LIN {X 0,Y 523.95,Z 619.34,A -85,B 0,C 180,E1 -4877.97,E2 -4877.97} C_VEL
LIN {X 0,Y 523.975,Z 619.339,A -85,B 0,C 180,E1 -4880.41,E2 -4880.41} C_VEL
LIN {X 0,Y 523.913,Z 619.349,A -85,B 0,C 180,E1 -4882.894,E2 -4882.894} C_VEL
LIN {X 0,Y 523.937,Z 619.342,A -85,B 0,C 180,E1 -4885.42,E2 -4885.42} C_VEL
LIN {X 0,Y 523.92,Z 619.339,A -85,B 0,C 180,E1 -4888.002,E2 -4888.002} C_VEL
LIN {X 0,Y 523.942,Z 619.344,A -85,B 0,C 180,E1 -4890.854,E2 -4890.854} C_VEL
LIN {X 0,Y 523.932,Z 619.34,A -85,B 0,C 180,E1 -4893.73,E2 -4893.73} C_VEL
LIN {X 0,Y 523.906,Z 619.346,A -85,B 0,C 180,E1 -4896.401,E2 -4896.401} C_VEL
LIN {X 0,Y 523.915,Z 619.351,A -85,B 0,C 180,E1 -4899.086,E2 -4899.086} C_VEL
LIN {X 0,Y 523.91,Z 619.344,A -85,B 0,C 180,E1 -4902.124,E2 -4902.124} C_VEL
LIN {X 0,Y 523.939,Z 619.346,A -85,B 0,C 180,E1 -4905.311,E2 -4905.311} C_VEL
LIN {X 0,Y 523.883,Z 619.351,A -85,B 0,C 180,E1 -4906.91,E2 -4906.91} C_VEL
LIN {X 0,Y 523.204,Z 619.439,A -85,B 0,C 180,E1 -4907.552,E2 -4907.552} C_VEL
LIN {X 0,Y 520.358,Z 619.789,A -85,B 0,C 180,E1 -4908.594,E2 -4908.594} C_VEL
LIN {X 0,Y 517.964,Z 620.093,A -85,B 0,C 180,E1 -4909.433,E2 -4909.433} C_VEL
LIN {X 0,Y 516.942,Z 620.215,A -85,B 0,C 180,E1 -4910.08,E2 -4910.08} C_VEL
LIN {X 0,Y 516.861,Z 620.224,A -85,B 0,C 180,E1 -4910.3,E2 -4910.3} C_VEL
LIN {X 0,Y 516.879,Z 620.229,A -85,B 0,C 180,E1 -4913.344,E2 -4913.344} C_VEL
LIN {X 0,Y 516.883,Z 620.22,A -85,B 0,C 180,E1 -4916.119,E2 -4916.119} C_VEL
LIN {X 0,Y 516.884,Z 620.224,A -85,B 0,C 180,E1 -4918.938,E2 -4918.938} C_VEL
LIN {X 0,Y 516.851,Z 620.232,A -85,B 0,C 180,E1 -4921.581,E2 -4921.581} C_VEL
LIN {X 0,Y 516.897,Z 620.309,A -85,B 0,C 180,E1 -4922.931,E2 -4922.931} C_VEL
LIN {X 0,Y 518.133,Z 627.417,A -85,B 0,C 180,E1 -4924.275,E2 -4924.275} C_VEL
LIN {X 0,Y 517.808,Z 639.497,A -85,B 0,C 180,E1 -4926.421,E2 -4926.421} C_VEL
LIN {X 0,Y 520.426,Z 652.346,A -85,B 0,C 180,E1 -4926.713,E2 -4926.713} C_VEL
LIN {X 0,Y 519.719,Z 775.501,A -85,B 0,C 180,E1 -4928.455,E2 -4928.455} C_VEL
LIN {X 0,Y 519.426,Z 789.891,A -85,B 0,C 180,E1 -4928.813,E2 -4928.813} C_VEL
LIN {X 0,Y 519.114,Z 803.721,A -85,B 0,C 180,E1 -4929.322,E2 -4929.322} C_VEL
LIN {X 0,Y 518.734,Z 817.355,A -85,B 0,C 180,E1 -4929.995,E2 -4929.995} C_VEL
LIN {X 0,Y 518.294,Z 830.118,A -85,B 0,C 180,E1 -4930.802,E2 -4930.802} C_VEL
LIN {X 0,Y 517.887,Z 841.924,A -85,B 0,C 180,E1 -4931.73,E2 -4931.73} C_VEL
LIN {X 0,Y 517.463,Z 853.262,A -85,B 0,C 180,E1 -4932.818,E2 -4932.818} C_VEL
LIN {X 0,Y 517.098,Z 863.506,A -85,B 0,C 180,E1 -4934.025,E2 -4934.025} C_VEL
LIN {X 0,Y 516.77,Z 873.237,A -85,B 0,C 180,E1 -4935.428,E2 -4935.428} C_VEL
LIN {X 0,Y 516.533,Z 881.108,A -85,B 0,C 180,E1 -4936.826,E2 -4936.826} C_VEL
LIN {X 0,Y 516.373,Z 887.392,A -85,B 0,C 180,E1 -4938.22,E2 -4938.22} C_VEL
LIN {X 0,Y 516.321,Z 891.674,A -85,B 0,C 180,E1 -4939.411,E2 -4939.411} C_VEL
LIN {X 0,Y 516.246,Z 895.077,A -85,B 0,C 180,E1 -4940.598,E2 -4940.598} C_VEL
LIN {X 0,Y 516.232,Z 898.246,A -85,B 0,C 180,E1 -4942.176,E2 -4942.176} C_VEL
LIN {X 0,Y 516.254,Z 900.019,A -85,B 0,C 180,E1 -4943.748,E2 -4943.748} C_VEL
LIN {X 0,Y 516.211,Z 900.451,A -85,B 0,C 180,E1 -4945.314,E2 -4945.314} C_VEL
LIN {X 0,Y 516.265,Z 899.556,A -85,B 0,C 180,E1 -4946.879,E2 -4946.879} C_VEL
LIN {X 0,Y 516.195,Z 897.325,A -85,B 0,C 180,E1 -4948.44,E2 -4948.44} C_VEL
LIN {X 0,Y 516.205,Z 893.711,A -85,B 0,C 180,E1 -4950,E2 -4950} C_VEL
LIN {X 0,Y 516.38,Z 890.026,A -85,B 0,C 180,E1 -4951.17,E2 -4951.17} C_VEL
LIN {X 0,Y 516.369,Z 885.463,A -85,B 0,C 180,E1 -4952.34,E2 -4952.34} C_VEL
LIN {X 0,Y 516.636,Z 878.835,A -85,B 0,C 180,E1 -4953.705,E2 -4953.705} C_VEL
LIN {X 0,Y 516.886,Z 870.62,A -85,B 0,C 180,E1 -4955.07,E2 -4955.07} C_VEL
LIN {X 0,Y 517.131,Z 862.132,A -85,B 0,C 180,E1 -4956.242,E2 -4956.242} C_VEL
LIN {X 0,Y 517.523,Z 851.815,A -85,B 0,C 180,E1 -4957.419,E2 -4957.419} C_VEL
LIN {X 0,Y 517.941,Z 840.432,A -85,B 0,C 180,E1 -4958.486,E2 -4958.486} C_VEL
LIN {X 0,Y 518.356,Z 829.005,A -85,B 0,C 180,E1 -4959.364,E2 -4959.364} C_VEL
LIN {X 0,Y 518.753,Z 816.473,A -85,B 0,C 180,E1 -4960.144,E2 -4960.144} C_VEL
LIN {X 0,Y 519.16,Z 803.502,A -85,B 0,C 180,E1 -4960.777,E2 -4960.777} C_VEL
LIN {X 0,Y 519.429,Z 789.513,A -85,B 0,C 180,E1 -4961.29,E2 -4961.29} C_VEL
LIN {X 0,Y 519.647,Z 775.805,A -85,B 0,C 180,E1 -4961.631,E2 -4961.631} C_VEL
LIN {X 0,Y 520.391,Z 652.06,A -85,B 0,C 180,E1 -4963.382,E2 -4963.382} C_VEL
LIN {X 0,Y 517.871,Z 639.491,A -85,B 0,C 180,E1 -4963.663,E2 -4963.663} C_VEL
LIN {X 0,Y 518.127,Z 626.693,A -85,B 0,C 180,E1 -4965.943,E2 -4965.943} C_VEL
LIN {X 0,Y 516.901,Z 620.224,A -85,B 0,C 180,E1 -4967.201,E2 -4967.201} C_VEL
LIN {X 0,Y 516.934,Z 620.221,A -85,B 0,C 180,E1 -4970.265,E2 -4970.265} C_VEL
LIN {X 0,Y 516.86,Z 620.226,A -85,B 0,C 180,E1 -4973.224,E2 -4973.224} C_VEL
LIN {X 0,Y 516.859,Z 620.226,A -85,B 0,C 180,E1 -4976.176,E2 -4976.176} C_VEL
LIN {X 0,Y 516.902,Z 620.22,A -85,B 0,C 180,E1 -4979.306,E2 -4979.306} C_VEL
LIN {X 0,Y 516.867,Z 620.227,A -85,B 0,C 180,E1 -4982.537,E2 -4982.537} C_VEL
LIN {X 0,Y 516.854,Z 620.226,A -85,B 0,C 180,E1 -4985.327,E2 -4985.327} C_VEL
LIN {X 0,Y 516.872,Z 620.227,A -85,B 0,C 180,E1 -4988.717,E2 -4988.717} C_VEL
LIN {X 0,Y 516.848,Z 620.224,A -85,B 0,C 180,E1 -4991.782,E2 -4991.782} C_VEL
LIN {X 0,Y 516.899,Z 620.225,A -85,B 0,C 180,E1 -4995.007,E2 -4995.007} C_VEL
LIN {X 0,Y 516.853,Z 620.224,A -85,B 0,C 180,E1 -4998.407,E2 -4998.407} C_VEL
LIN {X 0,Y 516.874,Z 620.221,A -85,B 0,C 180,E1 -5001.283,E2 -5001.283} C_VEL
LIN {X 0,Y 516.863,Z 620.22,A -85,B 0,C 180,E1 -5004.671,E2 -5004.671} C_VEL
LIN {X 0,Y 516.897,Z 620.223,A -85,B 0,C 180,E1 -5007.457,E2 -5007.457} C_VEL
LIN {X 0,Y 516.922,Z 620.213,A -85,B 0,C 180,E1 -5010.695,E2 -5010.695} C_VEL
LIN {X 0,Y 516.882,Z 620.221,A -85,B 0,C 180,E1 -5013.818,E2 -5013.818} C_VEL
LIN {X 0,Y 516.861,Z 620.22,A -85,B 0,C 180,E1 -5016.776,E2 -5016.776} C_VEL
LIN {X 0,Y 516.943,Z 620.216,A -85,B 0,C 180,E1 -5019.732,E2 -5019.732} C_VEL
LIN {X 0,Y 516.909,Z 620.21,A -85,B 0,C 180,E1 -5022.595,E2 -5022.595} C_VEL
LIN {X 0,Y 516.946,Z 620.213,A -85,B 0,C 180,E1 -5025.03,E2 -5025.03} C_VEL
LIN {X 0,Y 516.97,Z 620.207,A -85,B 0,C 180,E1 -5028.233,E2 -5028.233} C_VEL
LIN {X 0,Y 516.967,Z 620.211,A -85,B 0,C 180,E1 -5031.399,E2 -5031.399} C_VEL
LIN {X 0,Y 517.017,Z 620.202,A -85,B 0,C 180,E1 -5034.54,E2 -5034.54} C_VEL
LIN {X 0,Y 517.084,Z 620.201,A -85,B 0,C 180,E1 -5037.663,E2 -5037.663} C_VEL
LIN {X 0,Y 517.094,Z 620.19,A -85,B 0,C 180,E1 -5040.779,E2 -5040.779} C_VEL
LIN {X 0,Y 517.012,Z 620.204,A -85,B 0,C 180,E1 -5043.117,E2 -5043.117} C_VEL
LIN {X 0,Y 516.995,Z 620.209,A -85,B 0,C 180,E1 -5046.243,E2 -5046.243} C_VEL
LIN {X 0,Y 516.968,Z 620.21,A -85,B 0,C 180,E1 -5048.6,E2 -5048.6} C_VEL
LIN {X 0,Y 516.956,Z 620.215,A -85,B 0,C 180,E1 -5051.807,E2 -5051.807} C_VEL
LIN {X 0,Y 516.948,Z 620.209,A -85,B 0,C 180,E1 -5055.146,E2 -5055.146} C_VEL
LIN {X 0,Y 516.928,Z 620.22,A -85,B 0,C 180,E1 -5058.222,E2 -5058.222} C_VEL
LIN {X 0,Y 516.915,Z 620.216,A -85,B 0,C 180,E1 -5060.701,E2 -5060.701} C_VEL
LIN {X 0,Y 516.893,Z 620.224,A -85,B 0,C 180,E1 -5064.073,E2 -5064.073} C_VEL
LIN {X 0,Y 516.927,Z 620.215,A -85,B 0,C 180,E1 -5066.658,E2 -5066.658} C_VEL
LIN {X 0,Y 516.914,Z 620.216,A -85,B 0,C 180,E1 -5069.524,E2 -5069.524} C_VEL
LIN {X 0,Y 516.9,Z 620.223,A -85,B 0,C 180,E1 -5072.544,E2 -5072.544} C_VEL
LIN {X 0,Y 516.869,Z 620.221,A -85,B 0,C 180,E1 -5075.33,E2 -5075.33} C_VEL
LIN {X 0,Y 516.884,Z 620.222,A -85,B 0,C 180,E1 -5077.943,E2 -5077.943} C_VEL
LIN {X 0,Y 516.905,Z 620.222,A -85,B 0,C 180,E1 -5080.74,E2 -5080.74} C_VEL
LIN {X 0,Y 516.885,Z 620.22,A -85,B 0,C 180,E1 -5083.903,E2 -5083.903} C_VEL
LIN {X 0,Y 516.884,Z 620.222,A -85,B 0,C 180,E1 -5086.107,E2 -5086.107} C_VEL
LIN {X 0,Y 516.92,Z 620.221,A -85,B 0,C 180,E1 -5088.398,E2 -5088.398} C_VEL
LIN {X 0,Y 516.883,Z 620.222,A -85,B 0,C 180,E1 -5091.284,E2 -5091.284} C_VEL
LIN {X 0,Y 516.893,Z 620.222,A -85,B 0,C 180,E1 -5094.221,E2 -5094.221} C_VEL
LIN {X 0,Y 516.9,Z 620.223,A -85,B 0,C 180,E1 -5097.053,E2 -5097.053} C_VEL
LIN {X 0,Y 516.895,Z 620.221,A -85,B 0,C 180,E1 -5099.796,E2 -5099.796} C_VEL
LIN {X 0,Y 516.93,Z 620.22,A -85,B 0,C 180,E1 -5102.906,E2 -5102.906} C_VEL
LIN {X 0,Y 516.982,Z 620.308,A -85,B 0,C 180,E1 -5103.318,E2 -5103.318} C_VEL
LIN {X 0,Y 519.43,Z 632.291,A -85,B 0,C 180,E1 -5105.201,E2 -5105.201} C_VEL
LIN {X 0,Y 518.76,Z 652.815,A -85,B 0,C 180,E1 -5108.126,E2 -5108.126} C_VEL
LIN {X 0,Y 518.152,Z 675.928,A -85,B 0,C 180,E1 -5111.374,E2 -5111.374} C_VEL
LIN {X 0,Y 520.468,Z 690.281,A -85,B 0,C 180,E1 -5111.668,E2 -5111.668} C_VEL
LIN {X 0,Y 519.629,Z 814.592,A -85,B 0,C 180,E1 -5113.423,E2 -5113.423} C_VEL
LIN {X 0,Y 519.394,Z 829.055,A -85,B 0,C 180,E1 -5113.792,E2 -5113.792} C_VEL
LIN {X 0,Y 519.121,Z 842.489,A -85,B 0,C 180,E1 -5114.29,E2 -5114.29} C_VEL
LIN {X 0,Y 518.758,Z 854.701,A -85,B 0,C 180,E1 -5114.883,E2 -5114.883} C_VEL
LIN {X 0,Y 518.28,Z 867.555,A -85,B 0,C 180,E1 -5115.672,E2 -5115.672} C_VEL
LIN {X 0,Y 517.884,Z 879.251,A -85,B 0,C 180,E1 -5116.562,E2 -5116.562} C_VEL
LIN {X 0,Y 517.561,Z 888.983,A -85,B 0,C 180,E1 -5117.451,E2 -5117.451} C_VEL
LIN {X 0,Y 517.252,Z 899.705,A -85,B 0,C 180,E1 -5118.637,E2 -5118.637} C_VEL
LIN {X 0,Y 516.88,Z 908.555,A -85,B 0,C 180,E1 -5119.819,E2 -5119.819} C_VEL
LIN {X 0,Y 516.689,Z 915.917,A -85,B 0,C 180,E1 -5121.001,E2 -5121.001} C_VEL
LIN {X 0,Y 516.501,Z 922.054,A -85,B 0,C 180,E1 -5122.179,E2 -5122.179} C_VEL
LIN {X 0,Y 516.395,Z 928.568,A -85,B 0,C 180,E1 -5123.749,E2 -5123.749} C_VEL
LIN {X 0,Y 516.305,Z 932.38,A -85,B 0,C 180,E1 -5124.924,E2 -5124.924} C_VEL
LIN {X 0,Y 516.325,Z 935.316,A -85,B 0,C 180,E1 -5126.097,E2 -5126.097} C_VEL
LIN {X 0,Y 516.258,Z 938.002,A -85,B 0,C 180,E1 -5127.659,E2 -5127.659} C_VEL
LIN {X 0,Y 516.155,Z 939.334,A -85,B 0,C 180,E1 -5129.22,E2 -5129.22} C_VEL
LIN {X 0,Y 516.155,Z 939.334,A -85,B 0,C 180,E1 -5130.78,E2 -5130.78} C_VEL
LIN {X 0,Y 516.258,Z 938.005,A -85,B 0,C 180,E1 -5132.341,E2 -5132.341} C_VEL
LIN {X 0,Y 516.325,Z 935.32,A -85,B 0,C 180,E1 -5133.902,E2 -5133.902} C_VEL
LIN {X 0,Y 516.388,Z 931.201,A -85,B 0,C 180,E1 -5135.467,E2 -5135.467} C_VEL
LIN {X 0,Y 516.406,Z 925.526,A -85,B 0,C 180,E1 -5137.035,E2 -5137.035} C_VEL
LIN {X 0,Y 516.599,Z 919.127,A -85,B 0,C 180,E1 -5138.409,E2 -5138.409} C_VEL
LIN {X 0,Y 516.826,Z 911.174,A -85,B 0,C 180,E1 -5139.787,E2 -5139.787} C_VEL
LIN {X 0,Y 517.109,Z 902.852,A -85,B 0,C 180,E1 -5140.969,E2 -5140.969} C_VEL
LIN {X 0,Y 517.455,Z 892.433,A -85,B 0,C 180,E1 -5142.197,E2 -5142.197} C_VEL
LIN {X 0,Y 517.808,Z 881.609,A -85,B 0,C 180,E1 -5143.24,E2 -5143.24} C_VEL
LIN {X 0,Y 518.211,Z 870.422,A -85,B 0,C 180,E1 -5144.13,E2 -5144.13} C_VEL
LIN {X 0,Y 518.634,Z 858.246,A -85,B 0,C 180,E1 -5144.92,E2 -5144.92} C_VEL
LIN {X 0,Y 519.026,Z 844.741,A -85,B 0,C 180,E1 -5145.612,E2 -5145.612} C_VEL
LIN {X 0,Y 519.364,Z 830.319,A -85,B 0,C 180,E1 -5146.166,E2 -5146.166} C_VEL
LIN {X 0,Y 519.645,Z 815.731,A -85,B 0,C 180,E1 -5146.551,E2 -5146.551} C_VEL
LIN {X 0,Y 519.827,Z 787.602,A -85,B 0,C 180,E1 -5146.974,E2 -5146.974} C_VEL
LIN {X 0,Y 520.385,Z 688.558,A -85,B 0,C 180,E1 -5148.359,E2 -5148.359} C_VEL
LIN {X 0,Y 518.155,Z 675.916,A -85,B 0,C 180,E1 -5148.626,E2 -5148.626} C_VEL
LIN {X 0,Y 518.806,Z 651.311,A -85,B 0,C 180,E1 -5152.081,E2 -5152.081} C_VEL
LIN {X 0,Y 519.377,Z 633.721,A -85,B 0,C 180,E1 -5154.588,E2 -5154.588} C_VEL
LIN {X 0,Y 518.926,Z 629.314,A -85,B 0,C 180,E1 -5155.253,E2 -5155.253} C_VEL
LIN {X 0,Y 516.965,Z 620.217,A -85,B 0,C 180,E1 -5156.71,E2 -5156.71} C_VEL
LIN {X 0,Y 516.913,Z 620.223,A -85,B 0,C 180,E1 -5159.524,E2 -5159.524} C_VEL
LIN {X 0,Y 516.902,Z 620.218,A -85,B 0,C 180,E1 -5162.544,E2 -5162.544} C_VEL
LIN {X 0,Y 516.885,Z 620.224,A -85,B 0,C 180,E1 -5165.332,E2 -5165.332} C_VEL
LIN {X 0,Y 516.886,Z 620.221,A -85,B 0,C 180,E1 -5167.944,E2 -5167.944} C_VEL
LIN {X 0,Y 516.887,Z 620.218,A -85,B 0,C 180,E1 -5170.741,E2 -5170.741} C_VEL
LIN {X 0,Y 516.905,Z 620.219,A -85,B 0,C 180,E1 -5172.829,E2 -5172.829} C_VEL
LIN {X 0,Y 516.924,Z 620.215,A -85,B 0,C 180,E1 -5175.01,E2 -5175.01} C_VEL
LIN {X 0,Y 516.924,Z 620.212,A -85,B 0,C 180,E1 -5178.398,E2 -5178.398} C_VEL
LIN {X 0,Y 516.888,Z 620.224,A -85,B 0,C 180,E1 -5181.285,E2 -5181.285} C_VEL
LIN {X 0,Y 516.893,Z 620.22,A -85,B 0,C 180,E1 -5184.221,E2 -5184.221} C_VEL
LIN {X 0,Y 516.899,Z 620.217,A -85,B 0,C 180,E1 -5187.053,E2 -5187.053} C_VEL
LIN {X 0,Y 516.894,Z 620.22,A -85,B 0,C 180,E1 -5189.797,E2 -5189.797} C_VEL
LIN {X 0,Y 516.93,Z 620.214,A -85,B 0,C 180,E1 -5192.468,E2 -5192.468} C_VEL
LIN {X 0,Y 516.912,Z 620.215,A -85,B 0,C 180,E1 -5195.072,E2 -5195.072} C_VEL
LIN {X 0,Y 516.872,Z 620.224,A -85,B 0,C 180,E1 -5197.622,E2 -5197.622} C_VEL
LIN {X 0,Y 516.934,Z 620.219,A -85,B 0,C 180,E1 -5200.13,E2 -5200.13} C_VEL
LIN {X 0,Y 516.933,Z 620.214,A -85,B 0,C 180,E1 -5202.596,E2 -5202.596} C_VEL
LIN {X 0,Y 516.944,Z 620.211,A -85,B 0,C 180,E1 -5205.03,E2 -5205.03} C_VEL
LIN {X 0,Y 516.968,Z 620.217,A -85,B 0,C 180,E1 -5208.234,E2 -5208.234} C_VEL
LIN {X 0,Y 516.97,Z 620.206,A -85,B 0,C 180,E1 -5211.4,E2 -5211.4} C_VEL
LIN {X 0,Y 517.011,Z 620.207,A -85,B 0,C 180,E1 -5213.757,E2 -5213.757} C_VEL
LIN {X 0,Y 517.085,Z 620.195,A -85,B 0,C 180,E1 -5217.663,E2 -5217.663} C_VEL
LIN {X 0,Y 517.094,Z 620.195,A -85,B 0,C 180,E1 -5220.779,E2 -5220.779} C_VEL
LIN {X 0,Y 517.013,Z 620.204,A -85,B 0,C 180,E1 -5223.117,E2 -5223.117} C_VEL
LIN {X 0,Y 517.004,Z 620.207,A -85,B 0,C 180,E1 -5226.243,E2 -5226.243} C_VEL
LIN {X 0,Y 516.946,Z 620.21,A -85,B 0,C 180,E1 -5229.39,E2 -5229.39} C_VEL
LIN {X 0,Y 516.955,Z 620.21,A -85,B 0,C 180,E1 -5231.807,E2 -5231.807} C_VEL
LIN {X 0,Y 516.95,Z 620.212,A -85,B 0,C 180,E1 -5235.148,E2 -5235.148} C_VEL
LIN {X 0,Y 516.919,Z 620.218,A -85,B 0,C 180,E1 -5238.223,E2 -5238.223} C_VEL
LIN {X 0,Y 516.915,Z 620.223,A -85,B 0,C 180,E1 -5240.702,E2 -5240.702} C_VEL
LIN {X 0,Y 516.904,Z 620.216,A -85,B 0,C 180,E1 -5244.073,E2 -5244.073} C_VEL
LIN {X 0,Y 516.9,Z 620.224,A -85,B 0,C 180,E1 -5246.66,E2 -5246.66} C_VEL
LIN {X 0,Y 516.911,Z 620.212,A -85,B 0,C 180,E1 -5249.523,E2 -5249.523} C_VEL
LIN {X 0,Y 516.897,Z 620.222,A -85,B 0,C 180,E1 -5252.543,E2 -5252.543} C_VEL
LIN {X 0,Y 516.868,Z 620.226,A -85,B 0,C 180,E1 -5255.33,E2 -5255.33} C_VEL
LIN {X 0,Y 516.881,Z 620.22,A -85,B 0,C 180,E1 -5257.943,E2 -5257.943} C_VEL
LIN {X 0,Y 516.856,Z 620.225,A -85,B 0,C 180,E1 -5260.745,E2 -5260.745} C_VEL
LIN {X 0,Y 516.883,Z 620.221,A -85,B 0,C 180,E1 -5263.904,E2 -5263.904} C_VEL
LIN {X 0,Y 516.839,Z 620.23,A -85,B 0,C 180,E1 -5266.911,E2 -5266.911} C_VEL
LIN {X 0,Y 516.862,Z 620.229,A -85,B 0,C 180,E1 -5269.593,E2 -5269.593} C_VEL
LIN {X 0,Y 516.861,Z 620.224,A -85,B 0,C 180,E1 -5270.3,E2 -5270.3} C_VEL
LIN {X 0,Y 516.204,Z 620.312,A -85,B 0,C 180,E1 -5270.95,E2 -5270.95} C_VEL
LIN {X 0,Y 513.367,Z 620.666,A -85,B 0,C 180,E1 -5272.006,E2 -5272.006} C_VEL
LIN {X 0,Y 510.957,Z 620.967,A -85,B 0,C 180,E1 -5272.856,E2 -5272.856} C_VEL
LIN {X 0,Y 509.912,Z 621.094,A -85,B 0,C 180,E1 -5273.513,E2 -5273.513} C_VEL
LIN {X 0,Y 509.821,Z 621.102,A -85,B 0,C 180,E1 -5273.736,E2 -5273.736} C_VEL
LIN {X 0,Y 509.842,Z 621.097,A -85,B 0,C 180,E1 -5276.538,E2 -5276.538} C_VEL
LIN {X 0,Y 509.832,Z 621.106,A -85,B 0,C 180,E1 -5279.333,E2 -5279.333} C_VEL
LIN {X 0,Y 509.856,Z 621.101,A -85,B 0,C 180,E1 -5282.498,E2 -5282.498} C_VEL
LIN {X 0,Y 509.852,Z 621.138,A -85,B 0,C 180,E1 -5282.721,E2 -5282.721} C_VEL
LIN {X 0,Y 511.174,Z 628.426,A -85,B 0,C 180,E1 -5284.118,E2 -5284.118} C_VEL
LIN {X 0,Y 510.904,Z 639.791,A -85,B 0,C 180,E1 -5286.162,E2 -5286.162} C_VEL
LIN {X 0,Y 513.705,Z 653.774,A -85,B 0,C 180,E1 -5286.481,E2 -5286.481} C_VEL
LIN {X 0,Y 512.933,Z 776.04,A -85,B 0,C 180,E1 -5288.235,E2 -5288.235} C_VEL
LIN {X 0,Y 512.634,Z 790.304,A -85,B 0,C 180,E1 -5288.597,E2 -5288.597} C_VEL
LIN {X 0,Y 512.288,Z 803.914,A -85,B 0,C 180,E1 -5289.103,E2 -5289.103} C_VEL
LIN {X 0,Y 511.914,Z 816.371,A -85,B 0,C 180,E1 -5289.717,E2 -5289.717} C_VEL
LIN {X 0,Y 511.447,Z 829.379,A -85,B 0,C 180,E1 -5290.535,E2 -5290.535} C_VEL
LIN {X 0,Y 511.016,Z 841.139,A -85,B 0,C 180,E1 -5291.456,E2 -5291.456} C_VEL
LIN {X 0,Y 510.546,Z 852.851,A -85,B 0,C 180,E1 -5292.578,E2 -5292.578} C_VEL
LIN {X 0,Y 510.148,Z 863.255,A -85,B 0,C 180,E1 -5293.801,E2 -5293.801} C_VEL
LIN {X 0,Y 509.821,Z 871.8,A -85,B 0,C 180,E1 -5295.021,E2 -5295.021} C_VEL
LIN {X 0,Y 509.513,Z 879.914,A -85,B 0,C 180,E1 -5296.438,E2 -5296.438} C_VEL
LIN {X 0,Y 509.367,Z 885.606,A -85,B 0,C 180,E1 -5297.651,E2 -5297.651} C_VEL
LIN {X 0,Y 509.246,Z 891.531,A -85,B 0,C 180,E1 -5299.262,E2 -5299.262} C_VEL
LIN {X 0,Y 509.165,Z 894.947,A -85,B 0,C 180,E1 -5300.466,E2 -5300.466} C_VEL
LIN {X 0,Y 509.148,Z 898.154,A -85,B 0,C 180,E1 -5302.066,E2 -5302.066} C_VEL
LIN {X 0,Y 509.174,Z 899.977,A -85,B 0,C 180,E1 -5303.66,E2 -5303.66} C_VEL
LIN {X 0,Y 509.125,Z 900.465,A -85,B 0,C 180,E1 -5305.249,E2 -5305.249} C_VEL
LIN {X 0,Y 509.18,Z 899.625,A -85,B 0,C 180,E1 -5306.835,E2 -5306.835} C_VEL
LIN {X 0,Y 509.115,Z 897.467,A -85,B 0,C 180,E1 -5308.418,E2 -5308.418} C_VEL
LIN {X 0,Y 509.114,Z 893.951,A -85,B 0,C 180,E1 -5310,E2 -5310} C_VEL
LIN {X 0,Y 509.301,Z 890.359,A -85,B 0,C 180,E1 -5311.186,E2 -5311.186} C_VEL
LIN {X 0,Y 509.479,Z 884.133,A -85,B 0,C 180,E1 -5312.767,E2 -5312.767} C_VEL
LIN {X 0,Y 509.683,Z 877.218,A -85,B 0,C 180,E1 -5314.151,E2 -5314.151} C_VEL
LIN {X 0,Y 510.018,Z 868.671,A -85,B 0,C 180,E1 -5315.535,E2 -5315.535} C_VEL
LIN {X 0,Y 510.35,Z 859.752,A -85,B 0,C 180,E1 -5316.722,E2 -5316.722} C_VEL
LIN {X 0,Y 510.692,Z 848.985,A -85,B 0,C 180,E1 -5317.91,E2 -5317.91} C_VEL
LIN {X 0,Y 511.19,Z 838.032,A -85,B 0,C 180,E1 -5318.898,E2 -5318.898} C_VEL
LIN {X 0,Y 511.609,Z 825.99,A -85,B 0,C 180,E1 -5319.788,E2 -5319.788} C_VEL
LIN {X 0,Y 512.013,Z 814.452,A -85,B 0,C 180,E1 -5320.479,E2 -5320.479} C_VEL
LIN {X 0,Y 512.409,Z 800.705,A -85,B 0,C 180,E1 -5321.121,E2 -5321.121} C_VEL
LIN {X 0,Y 512.702,Z 787.022,A -85,B 0,C 180,E1 -5321.59,E2 -5321.59} C_VEL
LIN {X 0,Y 512.886,Z 772.902,A -85,B 0,C 180,E1 -5321.912,E2 -5321.912} C_VEL
LIN {X 0,Y 513.706,Z 653.591,A -85,B 0,C 180,E1 -5323.611,E2 -5323.611} C_VEL
LIN {X 0,Y 510.954,Z 639.664,A -85,B 0,C 180,E1 -5323.944,E2 -5323.944} C_VEL
LIN {X 0,Y 511.249,Z 628.452,A -85,B 0,C 180,E1 -5325.958,E2 -5325.958} C_VEL
LIN {X 0,Y 509.874,Z 621.099,A -85,B 0,C 180,E1 -5327.394,E2 -5327.394} C_VEL
LIN {X 0,Y 509.882,Z 621.101,A -85,B 0,C 180,E1 -5330.399,E2 -5330.399} C_VEL
LIN {X 0,Y 509.815,Z 621.102,A -85,B 0,C 180,E1 -5333.564,E2 -5333.564} C_VEL
LIN {X 0,Y 509.8,Z 621.108,A -85,B 0,C 180,E1 -5336.352,E2 -5336.352} C_VEL
LIN {X 0,Y 509.834,Z 621.105,A -85,B 0,C 180,E1 -5338.847,E2 -5338.847} C_VEL
LIN {X 0,Y 509.791,Z 621.104,A -85,B 0,C 180,E1 -5341.592,E2 -5341.592} C_VEL
LIN {X 0,Y 509.831,Z 621.102,A -85,B 0,C 180,E1 -5344.415,E2 -5344.415} C_VEL
LIN {X 0,Y 509.785,Z 621.107,A -85,B 0,C 180,E1 -5347.344,E2 -5347.344} C_VEL
LIN {X 0,Y 509.815,Z 621.096,A -85,B 0,C 180,E1 -5350.385,E2 -5350.385} C_VEL
LIN {X 0,Y 509.808,Z 621.101,A -85,B 0,C 180,E1 -5353.573,E2 -5353.573} C_VEL
LIN {X 0,Y 509.808,Z 621.102,A -85,B 0,C 180,E1 -5356.426,E2 -5356.426} C_VEL
LIN {X 0,Y 509.816,Z 621.102,A -85,B 0,C 180,E1 -5359.615,E2 -5359.615} C_VEL
LIN {X 0,Y 509.796,Z 621.097,A -85,B 0,C 180,E1 -5362.657,E2 -5362.657} C_VEL
LIN {X 0,Y 509.842,Z 621.098,A -85,B 0,C 180,E1 -5365.8,E2 -5365.8} C_VEL
LIN {X 0,Y 509.847,Z 621.097,A -85,B 0,C 180,E1 -5368.72,E2 -5368.72} C_VEL
LIN {X 0,Y 509.852,Z 621.099,A -85,B 0,C 180,E1 -5371.154,E2 -5371.154} C_VEL
LIN {X 0,Y 509.851,Z 621.097,A -85,B 0,C 180,E1 -5373.825,E2 -5373.825} C_VEL
LIN {X 0,Y 509.822,Z 621.095,A -85,B 0,C 180,E1 -5376.436,E2 -5376.436} C_VEL
LIN {X 0,Y 509.92,Z 621.089,A -85,B 0,C 180,E1 -5379.845,E2 -5379.845} C_VEL
LIN {X 0,Y 509.875,Z 621.091,A -85,B 0,C 180,E1 -5383.174,E2 -5383.174} C_VEL
LIN {X 0,Y 509.865,Z 621.102,A -85,B 0,C 180,E1 -5385.634,E2 -5385.634} C_VEL
LIN {X 0,Y 509.915,Z 621.085,A -85,B 0,C 180,E1 -5388.874,E2 -5388.874} C_VEL
LIN {X 0,Y 509.922,Z 621.09,A -85,B 0,C 180,E1 -5392.078,E2 -5392.078} C_VEL
LIN {X 0,Y 509.967,Z 621.081,A -85,B 0,C 180,E1 -5394.464,E2 -5394.464} C_VEL
LIN {X 0,Y 510.054,Z 621.076,A -85,B 0,C 180,E1 -5397.631,E2 -5397.631} C_VEL
LIN {X 0,Y 510.065,Z 621.066,A -85,B 0,C 180,E1 -5400.789,E2 -5400.789} C_VEL
LIN {X 0,Y 509.954,Z 621.083,A -85,B 0,C 180,E1 -5403.16,E2 -5403.16} C_VEL
LIN {X 0,Y 509.942,Z 621.086,A -85,B 0,C 180,E1 -5406.33,E2 -5406.33} C_VEL
LIN {X 0,Y 509.914,Z 621.088,A -85,B 0,C 180,E1 -5408.72,E2 -5408.72} C_VEL
LIN {X 0,Y 509.908,Z 621.095,A -85,B 0,C 180,E1 -5411.931,E2 -5411.931} C_VEL
LIN {X 0,Y 509.897,Z 621.088,A -85,B 0,C 180,E1 -5415.242,E2 -5415.242} C_VEL
LIN {X 0,Y 509.892,Z 621.098,A -85,B 0,C 180,E1 -5418.001,E2 -5418.001} C_VEL
LIN {X 0,Y 509.853,Z 621.094,A -85,B 0,C 180,E1 -5421.001,E2 -5421.001} C_VEL
LIN {X 0,Y 509.825,Z 621.098,A -85,B 0,C 180,E1 -5423.564,E2 -5423.564} C_VEL
LIN {X 0,Y 509.914,Z 621.093,A -85,B 0,C 180,E1 -5426.378,E2 -5426.378} C_VEL
LIN {X 0,Y 509.879,Z 621.094,A -85,B 0,C 180,E1 -5428.844,E2 -5428.844} C_VEL
LIN {X 0,Y 509.824,Z 621.099,A -85,B 0,C 180,E1 -5431.59,E2 -5431.59} C_VEL
LIN {X 0,Y 509.85,Z 621.104,A -85,B 0,C 180,E1 -5434.413,E2 -5434.413} C_VEL
LIN {X 0,Y 509.819,Z 621.099,A -85,B 0,C 180,E1 -5437.341,E2 -5437.341} C_VEL
LIN {X 0,Y 509.863,Z 621.101,A -85,B 0,C 180,E1 -5440.38,E2 -5440.38} C_VEL
LIN {X 0,Y 509.826,Z 621.1,A -85,B 0,C 180,E1 -5443.062,E2 -5443.062} C_VEL
LIN {X 0,Y 509.832,Z 621.098,A -85,B 0,C 180,E1 -5445.792,E2 -5445.792} C_VEL
LIN {X 0,Y 509.861,Z 621.103,A -85,B 0,C 180,E1 -5448.575,E2 -5448.575} C_VEL
LIN {X 0,Y 509.854,Z 621.096,A -85,B 0,C 180,E1 -5451.786,E2 -5451.786} C_VEL
LIN {X 0,Y 509.849,Z 621.105,A -85,B 0,C 180,E1 -5454.623,E2 -5454.623} C_VEL
LIN {X 0,Y 509.868,Z 621.095,A -85,B 0,C 180,E1 -5457.481,E2 -5457.481} C_VEL
LIN {X 0,Y 509.86,Z 621.1,A -85,B 0,C 180,E1 -5460.274,E2 -5460.274} C_VEL
LIN {X 0,Y 509.925,Z 621.206,A -85,B 0,C 180,E1 -5463.091,E2 -5463.091} C_VEL
LIN {X 0,Y 512.504,Z 633.266,A -85,B 0,C 180,E1 -5465.022,E2 -5465.022} C_VEL
LIN {X 0,Y 511.917,Z 651.073,A -85,B 0,C 180,E1 -5467.606,E2 -5467.606} C_VEL
LIN {X 0,Y 511.3,Z 670.083,A -85,B 0,C 180,E1 -5470.32,E2 -5470.32} C_VEL
LIN {X 0,Y 511.182,Z 675.688,A -85,B 0,C 180,E1 -5471.116,E2 -5471.116} C_VEL
LIN {X 0,Y 513.717,Z 690.981,A -85,B 0,C 180,E1 -5471.433,E2 -5471.433} C_VEL
LIN {X 0,Y 512.827,Z 814.311,A -85,B 0,C 180,E1 -5473.197,E2 -5473.197} C_VEL
LIN {X 0,Y 512.574,Z 828.954,A -85,B 0,C 180,E1 -5473.577,E2 -5473.577} C_VEL
LIN {X 0,Y 512.257,Z 842.212,A -85,B 0,C 180,E1 -5474.074,E2 -5474.074} C_VEL
LIN {X 0,Y 511.865,Z 854.425,A -85,B 0,C 180,E1 -5474.674,E2 -5474.674} C_VEL
LIN {X 0,Y 511.348,Z 867.279,A -85,B 0,C 180,E1 -5475.473,E2 -5475.473} C_VEL
LIN {X 0,Y 510.951,Z 878.977,A -85,B 0,C 180,E1 -5476.376,E2 -5476.376} C_VEL
LIN {X 0,Y 510.545,Z 889.752,A -85,B 0,C 180,E1 -5477.383,E2 -5477.383} C_VEL
LIN {X 0,Y 510.223,Z 899.511,A -85,B 0,C 180,E1 -5478.479,E2 -5478.479} C_VEL
LIN {X 0,Y 509.852,Z 908.425,A -85,B 0,C 180,E1 -5479.677,E2 -5479.677} C_VEL
LIN {X 0,Y 509.629,Z 915.849,A -85,B 0,C 180,E1 -5480.875,E2 -5480.875} C_VEL
LIN {X 0,Y 509.45,Z 922.04,A -85,B 0,C 180,E1 -5482.071,E2 -5482.071} C_VEL
LIN {X 0,Y 509.348,Z 927.783,A -85,B 0,C 180,E1 -5483.443,E2 -5483.443} C_VEL
LIN {X 0,Y 509.238,Z 932.38,A -85,B 0,C 180,E1 -5484.853,E2 -5484.853} C_VEL
LIN {X 0,Y 509.219,Z 935.315,A -85,B 0,C 180,E1 -5486.043,E2 -5486.043} C_VEL
LIN {X 0,Y 509.158,Z 938.003,A -85,B 0,C 180,E1 -5487.627,E2 -5487.627} C_VEL
LIN {X 0,Y 509.069,Z 939.334,A -85,B 0,C 180,E1 -5489.209,E2 -5489.209} C_VEL
LIN {X 0,Y 509.069,Z 939.334,A -85,B 0,C 180,E1 -5490.791,E2 -5490.791} C_VEL
LIN {X 0,Y 509.158,Z 938.006,A -85,B 0,C 180,E1 -5492.373,E2 -5492.373} C_VEL
LIN {X 0,Y 509.219,Z 935.32,A -85,B 0,C 180,E1 -5493.957,E2 -5493.957} C_VEL
LIN {X 0,Y 509.3,Z 931.201,A -85,B 0,C 180,E1 -5495.543,E2 -5495.543} C_VEL
LIN {X 0,Y 509.329,Z 925.526,A -85,B 0,C 180,E1 -5497.134,E2 -5497.134} C_VEL
LIN {X 0,Y 509.553,Z 919.087,A -85,B 0,C 180,E1 -5498.527,E2 -5498.527} C_VEL
LIN {X 0,Y 509.762,Z 911.063,A -85,B 0,C 180,E1 -5499.924,E2 -5499.924} C_VEL
LIN {X 0,Y 510.094,Z 902.677,A -85,B 0,C 180,E1 -5501.121,E2 -5501.121} C_VEL
LIN {X 0,Y 510.442,Z 892.508,A -85,B 0,C 180,E1 -5502.331,E2 -5502.331} C_VEL
LIN {X 0,Y 510.838,Z 881.327,A -85,B 0,C 180,E1 -5503.424,E2 -5503.424} C_VEL
LIN {X 0,Y 511.264,Z 870.139,A -85,B 0,C 180,E1 -5504.326,E2 -5504.326} C_VEL
LIN {X 0,Y 511.733,Z 857.962,A -85,B 0,C 180,E1 -5505.126,E2 -5505.126} C_VEL
LIN {X 0,Y 512.162,Z 844.457,A -85,B 0,C 180,E1 -5505.827,E2 -5505.827} C_VEL
LIN {X 0,Y 512.534,Z 830.117,A -85,B 0,C 180,E1 -5506.385,E2 -5506.385} C_VEL
LIN {X 0,Y 512.835,Z 815.442,A -85,B 0,C 180,E1 -5506.777,E2 -5506.777} C_VEL
LIN {X 0,Y 513.047,Z 787.309,A -85,B 0,C 180,E1 -5507.206,E2 -5507.206} C_VEL
LIN {X 0,Y 513.666,Z 689.639,A -85,B 0,C 180,E1 -5508.588,E2 -5508.588} C_VEL
LIN {X 0,Y 511.185,Z 675.612,A -85,B 0,C 180,E1 -5508.891,E2 -5508.891} C_VEL
LIN {X 0,Y 511.868,Z 652.505,A -85,B 0,C 180,E1 -5512.184,E2 -5512.184} C_VEL
LIN {X 0,Y 512.494,Z 634.961,A -85,B 0,C 180,E1 -5514.723,E2 -5514.723} C_VEL
LIN {X 0,Y 511.948,Z 630.535,A -85,B 0,C 180,E1 -5515.404,E2 -5515.404} C_VEL
LIN {X 0,Y 509.916,Z 621.095,A -85,B 0,C 180,E1 -5516.928,E2 -5516.928} C_VEL
LIN {X 0,Y 509.858,Z 621.099,A -85,B 0,C 180,E1 -5519.751,E2 -5519.751} C_VEL
LIN {X 0,Y 509.878,Z 621.094,A -85,B 0,C 180,E1 -5522.775,E2 -5522.775} C_VEL
LIN {X 0,Y 509.844,Z 621.102,A -85,B 0,C 180,E1 -5525.581,E2 -5525.581} C_VEL
LIN {X 0,Y 509.853,Z 621.095,A -85,B 0,C 180,E1 -5528.338,E2 -5528.338} C_VEL
LIN {X 0,Y 509.86,Z 621.101,A -85,B 0,C 180,E1 -5531.425,E2 -5531.425} C_VEL
LIN {X 0,Y 509.858,Z 621.093,A -85,B 0,C 180,E1 -5534.668,E2 -5534.668} C_VEL
LIN {X 0,Y 509.863,Z 621.094,A -85,B 0,C 180,E1 -5538.103,E2 -5538.103} C_VEL
LIN {X 0,Y 509.861,Z 621.095,A -85,B 0,C 180,E1 -5540.649,E2 -5540.649} C_VEL
LIN {X 0,Y 509.837,Z 621.1,A -85,B 0,C 180,E1 -5543.648,E2 -5543.648} C_VEL
LIN {X 0,Y 509.864,Z 621.093,A -85,B 0,C 180,E1 -5546.54,E2 -5546.54} C_VEL
LIN {X 0,Y 509.848,Z 621.09,A -85,B 0,C 180,E1 -5549.335,E2 -5549.335} C_VEL
LIN {X 0,Y 509.896,Z 621.095,A -85,B 0,C 180,E1 -5552.055,E2 -5552.055} C_VEL
LIN {X 0,Y 509.879,Z 621.091,A -85,B 0,C 180,E1 -5554.704,E2 -5554.704} C_VEL
LIN {X 0,Y 509.838,Z 621.098,A -85,B 0,C 180,E1 -5557.455,E2 -5557.455} C_VEL
LIN {X 0,Y 509.919,Z 621.094,A -85,B 0,C 180,E1 -5559.845,E2 -5559.845} C_VEL
LIN {X 0,Y 509.889,Z 621.09,A -85,B 0,C 180,E1 -5563.175,E2 -5563.175} C_VEL
LIN {X 0,Y 509.866,Z 621.096,A -85,B 0,C 180,E1 -5565.634,E2 -5565.634} C_VEL
LIN {X 0,Y 509.916,Z 621.088,A -85,B 0,C 180,E1 -5568.875,E2 -5568.875} C_VEL
LIN {X 0,Y 509.953,Z 621.088,A -85,B 0,C 180,E1 -5572.079,E2 -5572.079} C_VEL
LIN {X 0,Y 509.983,Z 621.082,A -85,B 0,C 180,E1 -5574.465,E2 -5574.465} C_VEL
LIN {X 0,Y 510.056,Z 621.071,A -85,B 0,C 180,E1 -5577.631,E2 -5577.631} C_VEL
LIN {X 0,Y 510.064,Z 621.07,A -85,B 0,C 180,E1 -5580.79,E2 -5580.79} C_VEL
LIN {X 0,Y 509.955,Z 621.083,A -85,B 0,C 180,E1 -5583.16,E2 -5583.16} C_VEL
LIN {X 0,Y 509.956,Z 621.086,A -85,B 0,C 180,E1 -5586.33,E2 -5586.33} C_VEL
LIN {X 0,Y 509.913,Z 621.092,A -85,B 0,C 180,E1 -5588.721,E2 -5588.721} C_VEL
LIN {X 0,Y 509.907,Z 621.089,A -85,B 0,C 180,E1 -5591.932,E2 -5591.932} C_VEL
LIN {X 0,Y 509.897,Z 621.089,A -85,B 0,C 180,E1 -5595.242,E2 -5595.242} C_VEL
LIN {X 0,Y 509.869,Z 621.094,A -85,B 0,C 180,E1 -5597.994,E2 -5597.994} C_VEL
LIN {X 0,Y 509.889,Z 621.093,A -85,B 0,C 180,E1 -5600.402,E2 -5600.402} C_VEL
LIN {X 0,Y 509.831,Z 621.096,A -85,B 0,C 180,E1 -5603.564,E2 -5603.564} C_VEL
LIN {X 0,Y 509.881,Z 621.095,A -85,B 0,C 180,E1 -5606.371,E2 -5606.371} C_VEL
LIN {X 0,Y 509.86,Z 621.089,A -85,B 0,C 180,E1 -5609.726,E2 -5609.726} C_VEL
LIN {X 0,Y 509.869,Z 621.1,A -85,B 0,C 180,E1 -5612.773,E2 -5612.773} C_VEL
LIN {X 0,Y 509.828,Z 621.1,A -85,B 0,C 180,E1 -5615.579,E2 -5615.579} C_VEL
LIN {X 0,Y 509.851,Z 621.097,A -85,B 0,C 180,E1 -5618.338,E2 -5618.338} C_VEL
LIN {X 0,Y 509.834,Z 621.102,A -85,B 0,C 180,E1 -5621.428,E2 -5621.428} C_VEL
LIN {X 0,Y 509.842,Z 621.1,A -85,B 0,C 180,E1 -5624.67,E2 -5624.67} C_VEL
LIN {X 0,Y 509.794,Z 621.109,A -85,B 0,C 180,E1 -5627.506,E2 -5627.506} C_VEL
LIN {X 0,Y 509.835,Z 621.101,A -85,B 0,C 180,E1 -5630.646,E2 -5630.646} C_VEL
LIN {X 0,Y 509.821,Z 621.102,A -85,B 0,C 180,E1 -5633.736,E2 -5633.736} C_VEL
LIN {X 0,Y 509.147,Z 621.184,A -85,B 0,C 180,E1 -5634.395,E2 -5634.395} C_VEL
LIN {X 0,Y 506.317,Z 621.544,A -85,B 0,C 180,E1 -5635.467,E2 -5635.467} C_VEL
LIN {X 0,Y 503.923,Z 621.839,A -85,B 0,C 180,E1 -5636.33,E2 -5636.33} C_VEL
LIN {X 0,Y 502.881,Z 621.965,A -85,B 0,C 180,E1 -5636.997,E2 -5636.997} C_VEL
LIN {X 0,Y 502.788,Z 621.976,A -85,B 0,C 180,E1 -5637.222,E2 -5637.222} C_VEL
LIN {X 0,Y 502.813,Z 621.978,A -85,B 0,C 180,E1 -5640.066,E2 -5640.066} C_VEL
LIN {X 0,Y 502.849,Z 622.137,A -85,B 0,C 180,E1 -5642.534,E2 -5642.534} C_VEL
LIN {X 0,Y 504.318,Z 630.644,A -85,B 0,C 180,E1 -5644.184,E2 -5644.184} C_VEL
LIN {X 0,Y 504.006,Z 640.099,A -85,B 0,C 180,E1 -5645.898,E2 -5645.898} C_VEL
LIN {X 0,Y 506.99,Z 654.639,A -85,B 0,C 180,E1 -5646.234,E2 -5646.234} C_VEL
LIN {X 0,Y 506.166,Z 776.533,A -85,B 0,C 180,E1 -5648.009,E2 -5648.009} C_VEL
LIN {X 0,Y 505.834,Z 790.983,A -85,B 0,C 180,E1 -5648.383,E2 -5648.383} C_VEL
LIN {X 0,Y 505.459,Z 804.883,A -85,B 0,C 180,E1 -5648.914,E2 -5648.914} C_VEL
LIN {X 0,Y 505.049,Z 817.185,A -85,B 0,C 180,E1 -5649.536,E2 -5649.536} C_VEL
LIN {X 0,Y 504.574,Z 830.09,A -85,B 0,C 180,E1 -5650.365,E2 -5650.365} C_VEL
LIN {X 0,Y 504.085,Z 841.77,A -85,B 0,C 180,E1 -5651.297,E2 -5651.297} C_VEL
LIN {X 0,Y 503.612,Z 852.433,A -85,B 0,C 180,E1 -5652.331,E2 -5652.331} C_VEL
LIN {X 0,Y 503.181,Z 862.975,A -85,B 0,C 180,E1 -5653.571,E2 -5653.571} C_VEL
LIN {X 0,Y 502.844,Z 871.482,A -85,B 0,C 180,E1 -5654.786,E2 -5654.786} C_VEL
LIN {X 0,Y 502.496,Z 879.834,A -85,B 0,C 180,E1 -5656.245,E2 -5656.245} C_VEL
LIN {X 0,Y 502.342,Z 885.579,A -85,B 0,C 180,E1 -5657.476,E2 -5657.476} C_VEL
LIN {X 0,Y 502.18,Z 891.589,A -85,B 0,C 180,E1 -5659.11,E2 -5659.11} C_VEL
LIN {X 0,Y 502.097,Z 895.037,A -85,B 0,C 180,E1 -5660.33,E2 -5660.33} C_VEL
LIN {X 0,Y 502.079,Z 898.324,A -85,B 0,C 180,E1 -5661.953,E2 -5661.953} C_VEL
LIN {X 0,Y 502.094,Z 900.229,A -85,B 0,C 180,E1 -5663.628,E2 -5663.628} C_VEL
LIN {X 0,Y 502.043,Z 900.734,A -85,B 0,C 180,E1 -5665.182,E2 -5665.182} C_VEL
LIN {X 0,Y 502.096,Z 899.956,A -85,B 0,C 180,E1 -5666.79,E2 -5666.79} C_VEL
LIN {X 0,Y 502.038,Z 897.863,A -85,B 0,C 180,E1 -5668.396,E2 -5668.396} C_VEL
LIN {X 0,Y 502.026,Z 894.406,A -85,B 0,C 180,E1 -5670,E2 -5670} C_VEL
LIN {X 0,Y 502.225,Z 890.876,A -85,B 0,C 180,E1 -5671.203,E2 -5671.203} C_VEL
LIN {X 0,Y 502.428,Z 884.714,A -85,B 0,C 180,E1 -5672.806,E2 -5672.806} C_VEL
LIN {X 0,Y 502.642,Z 877.872,A -85,B 0,C 180,E1 -5674.21,E2 -5674.21} C_VEL
LIN {X 0,Y 503.013,Z 869.405,A -85,B 0,C 180,E1 -5675.613,E2 -5675.613} C_VEL
LIN {X 0,Y 503.28,Z 862.18,A -85,B 0,C 180,E1 -5676.616,E2 -5676.616} C_VEL
LIN {X 0,Y 503.559,Z 853.923,A -85,B 0,C 180,E1 -5677.6,E2 -5677.6} C_VEL
LIN {X 0,Y 504.078,Z 842.575,A -85,B 0,C 180,E1 -5678.721,E2 -5678.721} C_VEL
LIN {X 0,Y 504.56,Z 831.487,A -85,B 0,C 180,E1 -5679.622,E2 -5679.622} C_VEL
LIN {X 0,Y 504.95,Z 819.428,A -85,B 0,C 180,E1 -5680.424,E2 -5680.424} C_VEL
LIN {X 0,Y 505.451,Z 806.017,A -85,B 0,C 180,E1 -5681.124,E2 -5681.124} C_VEL
LIN {X 0,Y 505.781,Z 791.967,A -85,B 0,C 180,E1 -5681.675,E2 -5681.675} C_VEL
LIN {X 0,Y 506.043,Z 778.094,A -85,B 0,C 180,E1 -5682.05,E2 -5682.05} C_VEL
LIN {X 0,Y 506.244,Z 752.41,A -85,B 0,C 180,E1 -5682.452,E2 -5682.452} C_VEL
LIN {X 0,Y 507.001,Z 654.584,A -85,B 0,C 180,E1 -5683.855,E2 -5683.855} C_VEL
LIN {X 0,Y 504.074,Z 639.949,A -85,B 0,C 180,E1 -5684.21,E2 -5684.21} C_VEL
LIN {X 0,Y 504.365,Z 630.326,A -85,B 0,C 180,E1 -5685.955,E2 -5685.955} C_VEL
LIN {X 0,Y 502.818,Z 621.979,A -85,B 0,C 180,E1 -5687.593,E2 -5687.593} C_VEL
LIN {X 0,Y 502.834,Z 621.98,A -85,B 0,C 180,E1 -5690.536,E2 -5690.536} C_VEL
LIN {X 0,Y 502.788,Z 621.981,A -85,B 0,C 180,E1 -5693.041,E2 -5693.041} C_VEL
LIN {X 0,Y 502.761,Z 621.981,A -85,B 0,C 180,E1 -5695.68,E2 -5695.68} C_VEL
LIN {X 0,Y 502.773,Z 621.983,A -85,B 0,C 180,E1 -5698.377,E2 -5698.377} C_VEL
LIN {X 0,Y 502.767,Z 621.984,A -85,B 0,C 180,E1 -5701.145,E2 -5701.145} C_VEL
LIN {X 0,Y 502.78,Z 621.977,A -85,B 0,C 180,E1 -5703.996,E2 -5703.996} C_VEL
LIN {X 0,Y 502.74,Z 621.987,A -85,B 0,C 180,E1 -5707.171,E2 -5707.171} C_VEL
LIN {X 0,Y 502.772,Z 621.971,A -85,B 0,C 180,E1 -5710.017,E2 -5710.017} C_VEL
LIN {X 0,Y 502.749,Z 621.985,A -85,B 0,C 180,E1 -5713.234,E2 -5713.234} C_VEL
LIN {X 0,Y 502.781,Z 621.978,A -85,B 0,C 180,E1 -5715.66,E2 -5715.66} C_VEL
LIN {X 0,Y 502.766,Z 621.986,A -85,B 0,C 180,E1 -5719.012,E2 -5719.012} C_VEL
LIN {X 0,Y 502.766,Z 621.97,A -85,B 0,C 180,E1 -5722.043,E2 -5722.043} C_VEL
LIN {X 0,Y 502.794,Z 621.976,A -85,B 0,C 180,E1 -5725.033,E2 -5725.033} C_VEL
LIN {X 0,Y 502.785,Z 621.976,A -85,B 0,C 180,E1 -5727.915,E2 -5727.915} C_VEL
LIN {X 0,Y 502.815,Z 621.97,A -85,B 0,C 180,E1 -5730.711,E2 -5730.711} C_VEL
LIN {X 0,Y 502.777,Z 621.983,A -85,B 0,C 180,E1 -5733.46,E2 -5733.46} C_VEL
LIN {X 0,Y 502.77,Z 621.974,A -85,B 0,C 180,E1 -5736.085,E2 -5736.085} C_VEL
LIN {X 0,Y 502.787,Z 621.976,A -85,B 0,C 180,E1 -5738.689,E2 -5738.689} C_VEL
LIN {X 0,Y 502.829,Z 621.975,A -85,B 0,C 180,E1 -5741.248,E2 -5741.248} C_VEL
LIN {X 0,Y 502.852,Z 621.966,A -85,B 0,C 180,E1 -5744.6,E2 -5744.6} C_VEL
LIN {X 0,Y 502.88,Z 621.963,A -85,B 0,C 180,E1 -5748.039,E2 -5748.039} C_VEL
LIN {X 0,Y 502.871,Z 621.964,A -85,B 0,C 180,E1 -5751.156,E2 -5751.156} C_VEL
LIN {X 0,Y 502.92,Z 621.959,A -85,B 0,C 180,E1 -5754.386,E2 -5754.386} C_VEL
LIN {X 0,Y 503.022,Z 621.952,A -85,B 0,C 180,E1 -5757.598,E2 -5757.598} C_VEL
LIN {X 0,Y 503.014,Z 621.944,A -85,B 0,C 180,E1 -5760.8,E2 -5760.8} C_VEL
LIN {X 0,Y 502.897,Z 621.963,A -85,B 0,C 180,E1 -5763.204,E2 -5763.204} C_VEL
LIN {X 0,Y 502.892,Z 621.964,A -85,B 0,C 180,E1 -5766.419,E2 -5766.419} C_VEL
LIN {X 0,Y 502.873,Z 621.965,A -85,B 0,C 180,E1 -5768.843,E2 -5768.843} C_VEL
LIN {X 0,Y 502.849,Z 621.975,A -85,B 0,C 180,E1 -5772.101,E2 -5772.101} C_VEL
LIN {X 0,Y 502.852,Z 621.966,A -85,B 0,C 180,E1 -5775.399,E2 -5775.399} C_VEL
LIN {X 0,Y 502.849,Z 621.975,A -85,B 0,C 180,E1 -5778.122,E2 -5778.122} C_VEL
LIN {X 0,Y 502.831,Z 621.972,A -85,B 0,C 180,E1 -5780.536,E2 -5780.536} C_VEL
LIN {X 0,Y 502.79,Z 621.973,A -85,B 0,C 180,E1 -5783.04,E2 -5783.04} C_VEL
LIN {X 0,Y 502.824,Z 621.972,A -85,B 0,C 180,E1 -5785.676,E2 -5785.676} C_VEL
LIN {X 0,Y 502.842,Z 621.976,A -85,B 0,C 180,E1 -5788.372,E2 -5788.372} C_VEL
LIN {X 0,Y 502.796,Z 621.974,A -85,B 0,C 180,E1 -5791.499,E2 -5791.499} C_VEL
LIN {X 0,Y 502.806,Z 621.977,A -85,B 0,C 180,E1 -5793.994,E2 -5793.994} C_VEL
LIN {X 0,Y 502.78,Z 621.977,A -85,B 0,C 180,E1 -5797.178,E2 -5797.178} C_VEL
LIN {X 0,Y 502.824,Z 621.973,A -85,B 0,C 180,E1 -5800.012,E2 -5800.012} C_VEL
LIN {X 0,Y 502.775,Z 621.978,A -85,B 0,C 180,E1 -5803.231,E2 -5803.231} C_VEL
LIN {X 0,Y 502.792,Z 621.975,A -85,B 0,C 180,E1 -5805.661,E2 -5805.661} C_VEL
LIN {X 0,Y 502.823,Z 621.976,A -85,B 0,C 180,E1 -5808.934,E2 -5808.934} C_VEL
LIN {X 0,Y 502.797,Z 621.977,A -85,B 0,C 180,E1 -5812.046,E2 -5812.046} C_VEL
LIN {X 0,Y 502.812,Z 621.979,A -85,B 0,C 180,E1 -5815.035,E2 -5815.035} C_VEL
LIN {X 0,Y 502.79,Z 621.977,A -85,B 0,C 180,E1 -5817.916,E2 -5817.916} C_VEL
LIN {X 0,Y 502.826,Z 621.979,A -85,B 0,C 180,E1 -5820.712,E2 -5820.712} C_VEL
LIN {X 0,Y 502.894,Z 622.109,A -85,B 0,C 180,E1 -5822.864,E2 -5822.864} C_VEL
LIN {X 0,Y 505.633,Z 635.343,A -85,B 0,C 180,E1 -5825.008,E2 -5825.008} C_VEL
LIN {X 0,Y 504.918,Z 655.201,A -85,B 0,C 180,E1 -5827.925,E2 -5827.925} C_VEL
LIN {X 0,Y 504.248,Z 675.352,A -85,B 0,C 180,E1 -5830.838,E2 -5830.838} C_VEL
LIN {X 0,Y 506.983,Z 691.834,A -85,B 0,C 180,E1 -5831.193,E2 -5831.193} C_VEL
LIN {X 0,Y 506.033,Z 814.031,A -85,B 0,C 180,E1 -5832.965,E2 -5832.965} C_VEL
LIN {X 0,Y 505.759,Z 828.59,A -85,B 0,C 180,E1 -5833.346,E2 -5833.346} C_VEL
LIN {X 0,Y 505.412,Z 841.936,A -85,B 0,C 180,E1 -5833.852,E2 -5833.852} C_VEL
LIN {X 0,Y 504.988,Z 854.149,A -85,B 0,C 180,E1 -5834.46,E2 -5834.46} C_VEL
LIN {X 0,Y 504.459,Z 867.005,A -85,B 0,C 180,E1 -5835.27,E2 -5835.27} C_VEL
LIN {X 0,Y 503.995,Z 878.701,A -85,B 0,C 180,E1 -5836.184,E2 -5836.184} C_VEL
LIN {X 0,Y 503.552,Z 889.519,A -85,B 0,C 180,E1 -5837.209,E2 -5837.209} C_VEL
LIN {X 0,Y 503.191,Z 899.235,A -85,B 0,C 180,E1 -5838.316,E2 -5838.316} C_VEL
LIN {X 0,Y 502.821,Z 908.151,A -85,B 0,C 180,E1 -5839.531,E2 -5839.531} C_VEL
LIN {X 0,Y 502.532,Z 916.7,A -85,B 0,C 180,E1 -5840.948,E2 -5840.948} C_VEL
LIN {X 0,Y 502.302,Z 923.591,A -85,B 0,C 180,E1 -5842.362,E2 -5842.362} C_VEL
LIN {X 0,Y 502.234,Z 928.345,A -85,B 0,C 180,E1 -5843.572,E2 -5843.572} C_VEL
LIN {X 0,Y 502.171,Z 932.195,A -85,B 0,C 180,E1 -5844.781,E2 -5844.781} C_VEL
LIN {X 0,Y 502.114,Z 935.161,A -85,B 0,C 180,E1 -5845.987,E2 -5845.987} C_VEL
LIN {X 0,Y 502.062,Z 937.877,A -85,B 0,C 180,E1 -5847.593,E2 -5847.593} C_VEL
LIN {X 0,Y 501.986,Z 939.221,A -85,B 0,C 180,E1 -5849.198,E2 -5849.198} C_VEL
LIN {X 0,Y 501.986,Z 939.221,A -85,B 0,C 180,E1 -5850.802,E2 -5850.802} C_VEL
LIN {X 0,Y 502.062,Z 937.879,A -85,B 0,C 180,E1 -5852.407,E2 -5852.407} C_VEL
LIN {X 0,Y 502.114,Z 935.165,A -85,B 0,C 180,E1 -5854.013,E2 -5854.013} C_VEL
LIN {X 0,Y 502.217,Z 931.003,A -85,B 0,C 180,E1 -5855.622,E2 -5855.622} C_VEL
LIN {X 0,Y 502.254,Z 925.267,A -85,B 0,C 180,E1 -5857.235,E2 -5857.235} C_VEL
LIN {X 0,Y 502.462,Z 918.808,A -85,B 0,C 180,E1 -5858.648,E2 -5858.648} C_VEL
LIN {X 0,Y 502.73,Z 910.785,A -85,B 0,C 180,E1 -5860.064,E2 -5860.064} C_VEL
LIN {X 0,Y 503.064,Z 902.397,A -85,B 0,C 180,E1 -5861.279,E2 -5861.279} C_VEL
LIN {X 0,Y 503.47,Z 891.661,A -85,B 0,C 180,E1 -5862.567,E2 -5862.567} C_VEL
LIN {X 0,Y 503.867,Z 881.045,A -85,B 0,C 180,E1 -5863.614,E2 -5863.614} C_VEL
LIN {X 0,Y 504.399,Z 868.426,A -85,B 0,C 180,E1 -5864.628,E2 -5864.628} C_VEL
LIN {X 0,Y 504.939,Z 855.907,A -85,B 0,C 180,E1 -5865.438,E2 -5865.438} C_VEL
LIN {X 0,Y 505.37,Z 843.041,A -85,B 0,C 180,E1 -5866.097,E2 -5866.097} C_VEL
LIN {X 0,Y 505.723,Z 829.123,A -85,B 0,C 180,E1 -5866.636,E2 -5866.636} C_VEL
LIN {X 0,Y 506.038,Z 815.154,A -85,B 0,C 180,E1 -5867.009,E2 -5867.009} C_VEL
LIN {X 0,Y 506.261,Z 788.806,A -85,B 0,C 180,E1 -5867.418,E2 -5867.418} C_VEL
LIN {X 0,Y 506.955,Z 690.732,A -85,B 0,C 180,E1 -5868.824,E2 -5868.824} C_VEL
LIN {X 0,Y 504.246,Z 675.327,A -85,B 0,C 180,E1 -5869.161,E2 -5869.161} C_VEL
LIN {X 0,Y 504.994,Z 652.242,A -85,B 0,C 180,E1 -5872.502,E2 -5872.502} C_VEL
LIN {X 0,Y 505.58,Z 635.309,A -85,B 0,C 180,E1 -5874.993,E2 -5874.993} C_VEL
LIN {X 0,Y 503.057,Z 622.854,A -85,B 0,C 180,E1 -5877.012,E2 -5877.012} C_VEL
LIN {X 0,Y 502.862,Z 621.973,A -85,B 0,C 180,E1 -5877.189,E2 -5877.189} C_VEL
LIN {X 0,Y 502.811,Z 621.975,A -85,B 0,C 180,E1 -5880.211,E2 -5880.211} C_VEL
LIN {X 0,Y 502.833,Z 621.973,A -85,B 0,C 180,E1 -5883.031,E2 -5883.031} C_VEL
LIN {X 0,Y 502.785,Z 621.977,A -85,B 0,C 180,E1 -5885.95,E2 -5885.95} C_VEL
LIN {X 0,Y 502.804,Z 621.977,A -85,B 0,C 180,E1 -5888.976,E2 -5888.976} C_VEL
LIN {X 0,Y 502.831,Z 621.972,A -85,B 0,C 180,E1 -5892.136,E2 -5892.136} C_VEL
LIN {X 0,Y 502.802,Z 621.981,A -85,B 0,C 180,E1 -5895.468,E2 -5895.468} C_VEL
LIN {X 0,Y 502.828,Z 621.97,A -85,B 0,C 180,E1 -5899.004,E2 -5899.004} C_VEL
LIN {X 0,Y 502.796,Z 621.971,A -85,B 0,C 180,E1 -5902.046,E2 -5902.046} C_VEL
LIN {X 0,Y 502.811,Z 621.973,A -85,B 0,C 180,E1 -5905.035,E2 -5905.035} C_VEL
LIN {X 0,Y 502.789,Z 621.971,A -85,B 0,C 180,E1 -5907.916,E2 -5907.916} C_VEL
LIN {X 0,Y 502.826,Z 621.969,A -85,B 0,C 180,E1 -5910.712,E2 -5910.712} C_VEL
LIN {X 0,Y 502.864,Z 621.968,A -85,B 0,C 180,E1 -5913.439,E2 -5913.439} C_VEL
LIN {X 0,Y 502.794,Z 621.979,A -85,B 0,C 180,E1 -5916.087,E2 -5916.087} C_VEL
LIN {X 0,Y 502.786,Z 621.976,A -85,B 0,C 180,E1 -5918.689,E2 -5918.689} C_VEL
LIN {X 0,Y 502.833,Z 621.969,A -85,B 0,C 180,E1 -5921.249,E2 -5921.249} C_VEL
LIN {X 0,Y 502.826,Z 621.975,A -85,B 0,C 180,E1 -5923.767,E2 -5923.767} C_VEL
LIN {X 0,Y 502.833,Z 621.975,A -85,B 0,C 180,E1 -5926.255,E2 -5926.255} C_VEL
LIN {X 0,Y 502.88,Z 621.966,A -85,B 0,C 180,E1 -5928.717,E2 -5928.717} C_VEL
LIN {X 0,Y 502.903,Z 621.964,A -85,B 0,C 180,E1 -5931.967,E2 -5931.967} C_VEL
LIN {X 0,Y 502.937,Z 621.961,A -85,B 0,C 180,E1 -5934.387,E2 -5934.387} C_VEL
LIN {X 0,Y 503.026,Z 621.946,A -85,B 0,C 180,E1 -5937.598,E2 -5937.598} C_VEL
LIN {X 0,Y 503.03,Z 621.949,A -85,B 0,C 180,E1 -5940,E2 -5940} C_VEL
LIN {X 0,Y 503.026,Z 621.954,A -85,B 0,C 180,E1 -5942.402,E2 -5942.402} C_VEL
LIN {X 0,Y 502.935,Z 621.954,A -85,B 0,C 180,E1 -5945.614,E2 -5945.614} C_VEL
LIN {X 0,Y 502.903,Z 621.964,A -85,B 0,C 180,E1 -5948.034,E2 -5948.034} C_VEL
LIN {X 0,Y 502.879,Z 621.964,A -85,B 0,C 180,E1 -5951.283,E2 -5951.283} C_VEL
LIN {X 0,Y 502.854,Z 621.973,A -85,B 0,C 180,E1 -5954.571,E2 -5954.571} C_VEL
LIN {X 0,Y 502.825,Z 621.971,A -85,B 0,C 180,E1 -5957.909,E2 -5957.909} C_VEL
LIN {X 0,Y 502.832,Z 621.974,A -85,B 0,C 180,E1 -5960.536,E2 -5960.536} C_VEL
LIN {X 0,Y 502.793,Z 621.978,A -85,B 0,C 180,E1 -5963.041,E2 -5963.041} C_VEL
LIN {X 0,Y 502.808,Z 621.973,A -85,B 0,C 180,E1 -5965.678,E2 -5965.678} C_VEL
LIN {X 0,Y 502.799,Z 621.972,A -85,B 0,C 180,E1 -5968.376,E2 -5968.376} C_VEL
LIN {X 0,Y 502.797,Z 621.98,A -85,B 0,C 180,E1 -5971.144,E2 -5971.144} C_VEL
LIN {X 0,Y 502.791,Z 621.973,A -85,B 0,C 180,E1 -5973.995,E2 -5973.995} C_VEL
LIN {X 0,Y 502.78,Z 621.984,A -85,B 0,C 180,E1 -5977.178,E2 -5977.178} C_VEL
LIN {X 0,Y 502.773,Z 621.974,A -85,B 0,C 180,E1 -5980.017,E2 -5980.017} C_VEL
LIN {X 0,Y 502.773,Z 621.977,A -85,B 0,C 180,E1 -5982.195,E2 -5982.195} C_VEL
LIN {X 0,Y 502.788,Z 621.979,A -85,B 0,C 180,E1 -5985.47,E2 -5985.47} C_VEL
LIN {X 0,Y 502.768,Z 621.981,A -85,B 0,C 180,E1 -5987.858,E2 -5987.858} C_VEL
LIN {X 0,Y 502.796,Z 621.982,A -85,B 0,C 180,E1 -5991.023,E2 -5991.023} C_VEL
LIN {X 0,Y 502.776,Z 621.977,A -85,B 0,C 180,E1 -5994.17,E2 -5994.17} C_VEL
LIN {X 0,Y 502.788,Z 621.976,A -85,B 0,C 180,E1 -5997.222,E2 -5997.222} C_VEL
LIN {X 0,Y 502.101,Z 622.064,A -85,B 0,C 180,E1 -5997.891,E2 -5997.891} C_VEL
LIN {X 0,Y 499.248,Z 622.422,A -85,B 0,C 180,E1 -5998.977,E2 -5998.977} C_VEL
LIN {X 0,Y 496.846,Z 622.723,A -85,B 0,C 180,E1 -5999.852,E2 -5999.852} C_VEL
LIN {X 0,Y 495.814,Z 622.848,A -85,B 0,C 180,E1 -6000.528,E2 -6000.528} C_VEL
LIN {X 0,Y 495.728,Z 622.859,A -85,B 0,C 180,E1 -6000.757,E2 -6000.757} C_VEL
LIN {X 0,Y 495.796,Z 622.983,A -85,B 0,C 180,E1 -6002.31,E2 -6002.31} C_VEL
LIN {X 0,Y 497.379,Z 631.657,A -85,B 0,C 180,E1 -6004.022,E2 -6004.022} C_VEL
LIN {X 0,Y 497.126,Z 640.339,A -85,B 0,C 180,E1 -6005.616,E2 -6005.616} C_VEL
LIN {X 0,Y 500.287,Z 655.753,A -85,B 0,C 180,E1 -6005.985,E2 -6005.985} C_VEL
LIN {X 0,Y 499.421,Z 776.229,A -85,B 0,C 180,E1 -6007.759,E2 -6007.759} C_VEL
LIN {X 0,Y 499.095,Z 790.714,A -85,B 0,C 180,E1 -6008.133,E2 -6008.133} C_VEL
LIN {X 0,Y 498.69,Z 804.189,A -85,B 0,C 180,E1 -6008.644,E2 -6008.644} C_VEL
LIN {X 0,Y 498.257,Z 816.201,A -85,B 0,C 180,E1 -6009.244,E2 -6009.244} C_VEL
LIN {X 0,Y 497.795,Z 827.901,A -85,B 0,C 180,E1 -6009.979,E2 -6009.979} C_VEL
LIN {X 0,Y 497.278,Z 840.021,A -85,B 0,C 180,E1 -6010.924,E2 -6010.924} C_VEL
LIN {X 0,Y 496.826,Z 850.041,A -85,B 0,C 180,E1 -6011.868,E2 -6011.868} C_VEL
LIN {X 0,Y 496.281,Z 861.028,A -85,B 0,C 180,E1 -6013.124,E2 -6013.124} C_VEL
LIN {X 0,Y 495.931,Z 870.054,A -85,B 0,C 180,E1 -6014.38,E2 -6014.38} C_VEL
LIN {X 0,Y 495.551,Z 878.649,A -85,B 0,C 180,E1 -6015.839,E2 -6015.839} C_VEL
LIN {X 0,Y 495.315,Z 885.537,A -85,B 0,C 180,E1 -6017.295,E2 -6017.295} C_VEL
LIN {X 0,Y 495.168,Z 890.258,A -85,B 0,C 180,E1 -6018.539,E2 -6018.539} C_VEL
LIN {X 0,Y 495.039,Z 895.125,A -85,B 0,C 180,E1 -6020.191,E2 -6020.191} C_VEL
LIN {X 0,Y 494.988,Z 898.478,A -85,B 0,C 180,E1 -6021.837,E2 -6021.837} C_VEL
LIN {X 0,Y 495.015,Z 900.421,A -85,B 0,C 180,E1 -6023.478,E2 -6023.478} C_VEL
LIN {X 0,Y 494.963,Z 901.02,A -85,B 0,C 180,E1 -6025.113,E2 -6025.113} C_VEL
LIN {X 0,Y 495.015,Z 900.297,A -85,B 0,C 180,E1 -6026.744,E2 -6026.744} C_VEL
LIN {X 0,Y 494.964,Z 898.26,A -85,B 0,C 180,E1 -6028.373,E2 -6028.373} C_VEL
LIN {X 0,Y 494.941,Z 894.861,A -85,B 0,C 180,E1 -6030,E2 -6030} C_VEL
LIN {X 0,Y 495.152,Z 891.384,A -85,B 0,C 180,E1 -6031.22,E2 -6031.22} C_VEL
LIN {X 0,Y 495.379,Z 885.296,A -85,B 0,C 180,E1 -6032.846,E2 -6032.846} C_VEL
LIN {X 0,Y 495.603,Z 878.526,A -85,B 0,C 180,E1 -6034.27,E2 -6034.27} C_VEL
LIN {X 0,Y 496.008,Z 870.139,A -85,B 0,C 180,E1 -6035.692,E2 -6035.692} C_VEL
LIN {X 0,Y 496.274,Z 863.009,A -85,B 0,C 180,E1 -6036.709,E2 -6036.709} C_VEL
LIN {X 0,Y 496.63,Z 854.041,A -85,B 0,C 180,E1 -6037.795,E2 -6037.795} C_VEL
LIN {X 0,Y 497.134,Z 843.647,A -85,B 0,C 180,E1 -6038.844,E2 -6038.844} C_VEL
LIN {X 0,Y 497.695,Z 831.332,A -85,B 0,C 180,E1 -6039.859,E2 -6039.859} C_VEL
LIN {X 0,Y 498.161,Z 819.162,A -85,B 0,C 180,E1 -6040.671,E2 -6040.671} C_VEL
LIN {X 0,Y 498.668,Z 805.606,A -85,B 0,C 180,E1 -6041.38,E2 -6041.38} C_VEL
LIN {X 0,Y 499.016,Z 791.32,A -85,B 0,C 180,E1 -6041.938,E2 -6041.938} C_VEL
LIN {X 0,Y 499.322,Z 776.978,A -85,B 0,C 180,E1 -6042.317,E2 -6042.317} C_VEL
LIN {X 0,Y 500.05,Z 693.382,A -85,B 0,C 180,E1 -6043.553,E2 -6043.553} C_VEL
LIN {X 0,Y 500.195,Z 654.842,A -85,B 0,C 180,E1 -6044.121,E2 -6044.121} C_VEL
LIN {X 0,Y 497.172,Z 640.252,A -85,B 0,C 180,E1 -6044.482,E2 -6044.482} C_VEL
LIN {X 0,Y 497.413,Z 631.439,A -85,B 0,C 180,E1 -6046.098,E2 -6046.098} C_VEL
LIN {X 0,Y 495.767,Z 622.857,A -85,B 0,C 180,E1 -6047.799,E2 -6047.799} C_VEL
LIN {X 0,Y 495.779,Z 622.858,A -85,B 0,C 180,E1 -6050.756,E2 -6050.756} C_VEL
LIN {X 0,Y 495.738,Z 622.857,A -85,B 0,C 180,E1 -6053.388,E2 -6053.388} C_VEL
LIN {X 0,Y 495.708,Z 622.861,A -85,B 0,C 180,E1 -6056.073,E2 -6056.073} C_VEL
LIN {X 0,Y 495.722,Z 622.862,A -85,B 0,C 180,E1 -6058.818,E2 -6058.818} C_VEL
LIN {X 0,Y 495.733,Z 622.856,A -85,B 0,C 180,E1 -6061.72,E2 -6061.72} C_VEL
LIN {X 0,Y 495.755,Z 622.859,A -85,B 0,C 180,E1 -6064.691,E2 -6064.691} C_VEL
LIN {X 0,Y 495.704,Z 622.859,A -85,B 0,C 180,E1 -6067.564,E2 -6067.564} C_VEL
LIN {X 0,Y 495.745,Z 622.846,A -85,B 0,C 180,E1 -6070.044,E2 -6070.044} C_VEL
LIN {X 0,Y 495.698,Z 622.866,A -85,B 0,C 180,E1 -6072.886,E2 -6072.886} C_VEL
LIN {X 0,Y 495.725,Z 622.855,A -85,B 0,C 180,E1 -6075.997,E2 -6075.997} C_VEL
LIN {X 0,Y 495.729,Z 622.86,A -85,B 0,C 180,E1 -6079.296,E2 -6079.296} C_VEL
LIN {X 0,Y 495.726,Z 622.852,A -85,B 0,C 180,E1 -6081.406,E2 -6081.406} C_VEL
LIN {X 0,Y 495.745,Z 622.848,A -85,B 0,C 180,E1 -6084.462,E2 -6084.462} C_VEL
LIN {X 0,Y 495.769,Z 622.856,A -85,B 0,C 180,E1 -6087.405,E2 -6087.405} C_VEL
LIN {X 0,Y 495.765,Z 622.846,A -85,B 0,C 180,E1 -6090.253,E2 -6090.253} C_VEL
LIN {X 0,Y 495.742,Z 622.861,A -85,B 0,C 180,E1 -6093.27,E2 -6093.27} C_VEL
LIN {X 0,Y 495.742,Z 622.849,A -85,B 0,C 180,E1 -6096.612,E2 -6096.612} C_VEL
LIN {X 0,Y 495.782,Z 622.855,A -85,B 0,C 180,E1 -6099.324,E2 -6099.324} C_VEL
LIN {X 0,Y 495.784,Z 622.845,A -85,B 0,C 180,E1 -6101.828,E2 -6101.828} C_VEL
LIN {X 0,Y 495.827,Z 622.841,A -85,B 0,C 180,E1 -6104.548,E2 -6104.548} C_VEL
LIN {X 0,Y 495.832,Z 622.842,A -85,B 0,C 180,E1 -6107.965,E2 -6107.965} C_VEL
LIN {X 0,Y 495.84,Z 622.838,A -85,B 0,C 180,E1 -6111.03,E2 -6111.03} C_VEL
LIN {X 0,Y 495.875,Z 622.837,A -85,B 0,C 180,E1 -6114.306,E2 -6114.306} C_VEL
LIN {X 0,Y 495.99,Z 622.827,A -85,B 0,C 180,E1 -6117.563,E2 -6117.563} C_VEL
LIN {X 0,Y 495.965,Z 622.822,A -85,B 0,C 180,E1 -6120.812,E2 -6120.812} C_VEL
LIN {X 0,Y 495.996,Z 622.823,A -85,B 0,C 180,E1 -6122.436,E2 -6122.436} C_VEL
LIN {X 0,Y 495.886,Z 622.84,A -85,B 0,C 180,E1 -6125.693,E2 -6125.693} C_VEL
LIN {X 0,Y 495.842,Z 622.841,A -85,B 0,C 180,E1 -6128.97,E2 -6128.97} C_VEL
LIN {X 0,Y 495.831,Z 622.85,A -85,B 0,C 180,E1 -6132.035,E2 -6132.035} C_VEL
LIN {X 0,Y 495.827,Z 622.841,A -85,B 0,C 180,E1 -6135.451,E2 -6135.451} C_VEL
LIN {X 0,Y 495.81,Z 622.849,A -85,B 0,C 180,E1 -6138.247,E2 -6138.247} C_VEL
LIN {X 0,Y 495.777,Z 622.849,A -85,B 0,C 180,E1 -6140.756,E2 -6140.756} C_VEL
LIN {X 0,Y 495.745,Z 622.851,A -85,B 0,C 180,E1 -6143.387,E2 -6143.387} C_VEL
LIN {X 0,Y 495.826,Z 622.843,A -85,B 0,C 180,E1 -6146.749,E2 -6146.749} C_VEL
LIN {X 0,Y 495.768,Z 622.852,A -85,B 0,C 180,E1 -6149.746,E2 -6149.746} C_VEL
LIN {X 0,Y 495.77,Z 622.855,A -85,B 0,C 180,E1 -6152.594,E2 -6152.594} C_VEL
LIN {X 0,Y 495.75,Z 622.853,A -85,B 0,C 180,E1 -6155.537,E2 -6155.537} C_VEL
LIN {X 0,Y 495.771,Z 622.853,A -85,B 0,C 180,E1 -6158.769,E2 -6158.769} C_VEL
LIN {X 0,Y 495.761,Z 622.851,A -85,B 0,C 180,E1 -6161.781,E2 -6161.781} C_VEL
LIN {X 0,Y 495.751,Z 622.853,A -85,B 0,C 180,E1 -6165.139,E2 -6165.139} C_VEL
LIN {X 0,Y 495.779,Z 622.852,A -85,B 0,C 180,E1 -6168.221,E2 -6168.221} C_VEL
LIN {X 0,Y 495.753,Z 622.853,A -85,B 0,C 180,E1 -6171.408,E2 -6171.408} C_VEL
LIN {X 0,Y 495.76,Z 622.858,A -85,B 0,C 180,E1 -6174.463,E2 -6174.463} C_VEL
LIN {X 0,Y 495.772,Z 622.852,A -85,B 0,C 180,E1 -6177.406,E2 -6177.406} C_VEL
LIN {X 0,Y 495.768,Z 622.856,A -85,B 0,C 180,E1 -6180.254,E2 -6180.254} C_VEL
LIN {X 0,Y 495.834,Z 622.966,A -85,B 0,C 180,E1 -6182.627,E2 -6182.627} C_VEL
LIN {X 0,Y 498.699,Z 636.362,A -85,B 0,C 180,E1 -6184.83,E2 -6184.83} C_VEL
LIN {X 0,Y 498.147,Z 652.026,A -85,B 0,C 180,E1 -6187.171,E2 -6187.171} C_VEL
LIN {X 0,Y 497.42,Z 670.984,A -85,B 0,C 180,E1 -6189.963,E2 -6189.963} C_VEL
LIN {X 0,Y 497.313,Z 675.088,A -85,B 0,C 180,E1 -6190.563,E2 -6190.563} C_VEL
LIN {X 0,Y 500.249,Z 692.78,A -85,B 0,C 180,E1 -6190.948,E2 -6190.948} C_VEL
LIN {X 0,Y 499.261,Z 813.751,A -85,B 0,C 180,E1 -6192.726,E2 -6192.726} C_VEL
LIN {X 0,Y 498.924,Z 828.115,A -85,B 0,C 180,E1 -6193.104,E2 -6193.104} C_VEL
LIN {X 0,Y 498.571,Z 841.659,A -85,B 0,C 180,E1 -6193.625,E2 -6193.625} C_VEL
LIN {X 0,Y 498.127,Z 853.874,A -85,B 0,C 180,E1 -6194.241,E2 -6194.241} C_VEL
LIN {X 0,Y 497.575,Z 866.73,A -85,B 0,C 180,E1 -6195.062,E2 -6195.062} C_VEL
LIN {X 0,Y 497.039,Z 878.426,A -85,B 0,C 180,E1 -6195.987,E2 -6195.987} C_VEL
LIN {X 0,Y 496.559,Z 889.244,A -85,B 0,C 180,E1 -6197.026,E2 -6197.026} C_VEL
LIN {X 0,Y 496.174,Z 899.172,A -85,B 0,C 180,E1 -6198.175,E2 -6198.175} C_VEL
LIN {X 0,Y 495.78,Z 907.877,A -85,B 0,C 180,E1 -6199.381,E2 -6199.381} C_VEL
LIN {X 0,Y 495.463,Z 916.425,A -85,B 0,C 180,E1 -6200.817,E2 -6200.817} C_VEL
LIN {X 0,Y 495.223,Z 923.317,A -85,B 0,C 180,E1 -6202.252,E2 -6202.252} C_VEL
LIN {X 0,Y 495.127,Z 929.034,A -85,B 0,C 180,E1 -6203.754,E2 -6203.754} C_VEL
LIN {X 0,Y 495.031,Z 932.996,A -85,B 0,C 180,E1 -6205.113,E2 -6205.113} C_VEL
LIN {X 0,Y 495.033,Z 936.422,A -85,B 0,C 180,E1 -6206.744,E2 -6206.744} C_VEL
LIN {X 0,Y 494.957,Z 938.446,A -85,B 0,C 180,E1 -6208.373,E2 -6208.373} C_VEL
LIN {X 0,Y 494.896,Z 939.116,A -85,B 0,C 180,E1 -6210,E2 -6210} C_VEL
LIN {X 0,Y 494.957,Z 938.447,A -85,B 0,C 180,E1 -6211.627,E2 -6211.627} C_VEL
LIN {X 0,Y 495.033,Z 936.424,A -85,B 0,C 180,E1 -6213.255,E2 -6213.255} C_VEL
LIN {X 0,Y 495.031,Z 932.995,A -85,B 0,C 180,E1 -6214.886,E2 -6214.886} C_VEL
LIN {X 0,Y 495.126,Z 929.031,A -85,B 0,C 180,E1 -6216.245,E2 -6216.245} C_VEL
LIN {X 0,Y 495.222,Z 923.309,A -85,B 0,C 180,E1 -6217.748,E2 -6217.748} C_VEL
LIN {X 0,Y 495.463,Z 916.417,A -85,B 0,C 180,E1 -6219.182,E2 -6219.182} C_VEL
LIN {X 0,Y 495.771,Z 907.864,A -85,B 0,C 180,E1 -6220.619,E2 -6220.619} C_VEL
LIN {X 0,Y 496.202,Z 898.052,A -85,B 0,C 180,E1 -6221.964,E2 -6221.964} C_VEL
LIN {X 0,Y 496.6,Z 888.147,A -85,B 0,C 180,E1 -6223.087,E2 -6223.087} C_VEL
LIN {X 0,Y 497.116,Z 877.227,A -85,B 0,C 180,E1 -6224.115,E2 -6224.115} C_VEL
LIN {X 0,Y 497.65,Z 865.281,A -85,B 0,C 180,E1 -6225.04,E2 -6225.04} C_VEL
LIN {X 0,Y 498.166,Z 852.065,A -85,B 0,C 180,E1 -6225.863,E2 -6225.863} C_VEL
LIN {X 0,Y 498.616,Z 839.008,A -85,B 0,C 180,E1 -6226.493,E2 -6226.493} C_VEL
LIN {X 0,Y 499.007,Z 824.789,A -85,B 0,C 180,E1 -6226.998,E2 -6226.998} C_VEL
LIN {X 0,Y 499.319,Z 810.952,A -85,B 0,C 180,E1 -6227.324,E2 -6227.324} C_VEL
LIN {X 0,Y 500.112,Z 691.095,A -85,B 0,C 180,E1 -6229.082,E2 -6229.082} C_VEL
LIN {X 0,Y 497.296,Z 675.04,A -85,B 0,C 180,E1 -6229.44,E2 -6229.44} C_VEL
LIN {X 0,Y 498.031,Z 654.905,A -85,B 0,C 180,E1 -6232.396,E2 -6232.396} C_VEL
LIN {X 0,Y 498.717,Z 637.374,A -85,B 0,C 180,E1 -6235.009,E2 -6235.009} C_VEL
LIN {X 0,Y 497.094,Z 628.581,A -85,B 0,C 180,E1 -6236.446,E2 -6236.446} C_VEL
LIN {X 0,Y 495.817,Z 622.851,A -85,B 0,C 180,E1 -6237.431,E2 -6237.431} C_VEL
LIN {X 0,Y 495.754,Z 622.856,A -85,B 0,C 180,E1 -6240.687,E2 -6240.687} C_VEL
LIN {X 0,Y 495.762,Z 622.855,A -85,B 0,C 180,E1 -6243.564,E2 -6243.564} C_VEL
LIN {X 0,Y 495.737,Z 622.854,A -85,B 0,C 180,E1 -6246.543,E2 -6246.543} C_VEL
LIN {X 0,Y 495.759,Z 622.855,A -85,B 0,C 180,E1 -6249.638,E2 -6249.638} C_VEL
LIN {X 0,Y 495.742,Z 622.854,A -85,B 0,C 180,E1 -6252.507,E2 -6252.507} C_VEL
LIN {X 0,Y 495.75,Z 622.854,A -85,B 0,C 180,E1 -6255.139,E2 -6255.139} C_VEL
LIN {X 0,Y 495.762,Z 622.849,A -85,B 0,C 180,E1 -6258.22,E2 -6258.22} C_VEL
LIN {X 0,Y 495.77,Z 622.854,A -85,B 0,C 180,E1 -6261.231,E2 -6261.231} C_VEL
LIN {X 0,Y 495.759,Z 622.851,A -85,B 0,C 180,E1 -6264.463,E2 -6264.463} C_VEL
LIN {X 0,Y 495.771,Z 622.853,A -85,B 0,C 180,E1 -6267.406,E2 -6267.406} C_VEL
LIN {X 0,Y 495.768,Z 622.851,A -85,B 0,C 180,E1 -6270.254,E2 -6270.254} C_VEL
LIN {X 0,Y 495.825,Z 622.843,A -85,B 0,C 180,E1 -6273.251,E2 -6273.251} C_VEL
LIN {X 0,Y 495.755,Z 622.858,A -85,B 0,C 180,E1 -6275.725,E2 -6275.725} C_VEL
LIN {X 0,Y 495.746,Z 622.855,A -85,B 0,C 180,E1 -6278.371,E2 -6278.371} C_VEL
LIN {X 0,Y 495.787,Z 622.846,A -85,B 0,C 180,E1 -6280.972,E2 -6280.972} C_VEL
LIN {X 0,Y 495.783,Z 622.85,A -85,B 0,C 180,E1 -6283.53,E2 -6283.53} C_VEL
LIN {X 0,Y 495.796,Z 622.851,A -85,B 0,C 180,E1 -6286.056,E2 -6286.056} C_VEL
LIN {X 0,Y 495.854,Z 622.842,A -85,B 0,C 180,E1 -6288.555,E2 -6288.555} C_VEL
LIN {X 0,Y 495.875,Z 622.837,A -85,B 0,C 180,E1 -6291.852,E2 -6291.852} C_VEL
LIN {X 0,Y 495.893,Z 622.84,A -85,B 0,C 180,E1 -6294.307,E2 -6294.307} C_VEL
LIN {X 0,Y 495.995,Z 622.822,A -85,B 0,C 180,E1 -6297.564,E2 -6297.564} C_VEL
LIN {X 0,Y 495.985,Z 622.823,A -85,B 0,C 180,E1 -6300.812,E2 -6300.812} C_VEL
LIN {X 0,Y 495.995,Z 622.83,A -85,B 0,C 180,E1 -6302.437,E2 -6302.437} C_VEL
LIN {X 0,Y 495.891,Z 622.831,A -85,B 0,C 180,E1 -6305.694,E2 -6305.694} C_VEL
LIN {X 0,Y 495.874,Z 622.841,A -85,B 0,C 180,E1 -6308.148,E2 -6308.148} C_VEL
LIN {X 0,Y 495.854,Z 622.838,A -85,B 0,C 180,E1 -6311.445,E2 -6311.445} C_VEL
LIN {X 0,Y 495.797,Z 622.85,A -85,B 0,C 180,E1 -6314.783,E2 -6314.783} C_VEL
LIN {X 0,Y 495.767,Z 622.851,A -85,B 0,C 180,E1 -6317.32,E2 -6317.32} C_VEL
LIN {X 0,Y 495.773,Z 622.847,A -85,B 0,C 180,E1 -6319.891,E2 -6319.891} C_VEL
LIN {X 0,Y 495.762,Z 622.855,A -85,B 0,C 180,E1 -6322.861,E2 -6322.861} C_VEL
LIN {X 0,Y 495.766,Z 622.851,A -85,B 0,C 180,E1 -6326.07,E2 -6326.07} C_VEL
LIN {X 0,Y 495.746,Z 622.85,A -85,B 0,C 180,E1 -6328.817,E2 -6328.817} C_VEL
LIN {X 0,Y 495.757,Z 622.852,A -85,B 0,C 180,E1 -6331.725,E2 -6331.725} C_VEL
LIN {X 0,Y 495.765,Z 622.853,A -85,B 0,C 180,E1 -6334.693,E2 -6334.693} C_VEL
LIN {X 0,Y 495.731,Z 622.857,A -85,B 0,C 180,E1 -6337.562,E2 -6337.562} C_VEL
LIN {X 0,Y 495.746,Z 622.85,A -85,B 0,C 180,E1 -6340.045,E2 -6340.045} C_VEL
LIN {X 0,Y 495.707,Z 622.863,A -85,B 0,C 180,E1 -6342.886,E2 -6342.886} C_VEL
LIN {X 0,Y 495.725,Z 622.856,A -85,B 0,C 180,E1 -6345.998,E2 -6345.998} C_VEL
LIN {X 0,Y 495.73,Z 622.865,A -85,B 0,C 180,E1 -6349.296,E2 -6349.296} C_VEL
LIN {X 0,Y 495.749,Z 622.861,A -85,B 0,C 180,E1 -6351.408,E2 -6351.408} C_VEL
LIN {X 0,Y 495.748,Z 622.852,A -85,B 0,C 180,E1 -6354.462,E2 -6354.462} C_VEL
LIN {X 0,Y 495.754,Z 622.851,A -85,B 0,C 180,E1 -6357.405,E2 -6357.405} C_VEL
LIN {X 0,Y 495.76,Z 622.855,A -85,B 0,C 180,E1 -6360.253,E2 -6360.253} C_VEL
LIN {X 0,Y 495.728,Z 622.859,A -85,B 0,C 180,E1 -6360.757,E2 -6360.757} C_VEL
LIN {X 0,Y 495.081,Z 623.097,A -85,B 0,C 180,E1 -6361.216,E2 -6361.216} C_VEL
LIN {X 0,Y 492.445,Z 624.384,A -85,B 0,C 180,E1 -6361.932,E2 -6361.932} C_VEL
LIN {X 0,Y 490.012,Z 626.701,A -85,B 0,C 180,E1 -6362.622,E2 -6362.622} C_VEL
LIN {X 0,Y 489.684,Z 628.569,A -85,B 0,C 180,E1 -6363.036,E2 -6363.036} C_VEL
LIN {X 0,Y 490.497,Z 633.882,A -85,B 0,C 180,E1 -6364.087,E2 -6364.087} C_VEL
LIN {X 0,Y 490.283,Z 640.903,A -85,B 0,C 180,E1 -6365.348,E2 -6365.348} C_VEL
LIN {X 0,Y 493.564,Z 656.154,A -85,B 0,C 180,E1 -6365.717,E2 -6365.717} C_VEL
LIN {X 0,Y 492.677,Z 776.389,A -85,B 0,C 180,E1 -6367.513,E2 -6367.513} C_VEL
LIN {X 0,Y 492.384,Z 790.154,A -85,B 0,C 180,E1 -6367.866,E2 -6367.866} C_VEL
LIN {X 0,Y 491.896,Z 804.326,A -85,B 0,C 180,E1 -6368.404,E2 -6368.404} C_VEL
LIN {X 0,Y 491.403,Z 817.016,A -85,B 0,C 180,E1 -6369.05,E2 -6369.05} C_VEL
LIN {X 0,Y 490.878,Z 830.062,A -85,B 0,C 180,E1 -6369.903,E2 -6369.903} C_VEL
LIN {X 0,Y 490.315,Z 841.744,A -85,B 0,C 180,E1 -6370.851,E2 -6370.851} C_VEL
LIN {X 0,Y 489.822,Z 851.6,A -85,B 0,C 180,E1 -6371.816,E2 -6371.816} C_VEL
LIN {X 0,Y 489.269,Z 862.372,A -85,B 0,C 180,E1 -6373.09,E2 -6373.09} C_VEL
LIN {X 0,Y 488.875,Z 871.493,A -85,B 0,C 180,E1 -6374.406,E2 -6374.406} C_VEL
LIN {X 0,Y 488.483,Z 879.654,A -85,B 0,C 180,E1 -6375.843,E2 -6375.843} C_VEL
LIN {X 0,Y 488.272,Z 885.494,A -85,B 0,C 180,E1 -6377.109,E2 -6377.109} C_VEL
LIN {X 0,Y 488.105,Z 890.283,A -85,B 0,C 180,E1 -6378.371,E2 -6378.371} C_VEL
LIN {X 0,Y 487.99,Z 895.214,A -85,B 0,C 180,E1 -6380.048,E2 -6380.048} C_VEL
LIN {X 0,Y 487.915,Z 898.626,A -85,B 0,C 180,E1 -6381.718,E2 -6381.718} C_VEL
LIN {X 0,Y 487.934,Z 900.633,A -85,B 0,C 180,E1 -6383.383,E2 -6383.383} C_VEL
LIN {X 0,Y 487.887,Z 901.299,A -85,B 0,C 180,E1 -6385.042,E2 -6385.042} C_VEL
LIN {X 0,Y 487.936,Z 900.638,A -85,B 0,C 180,E1 -6386.697,E2 -6386.697} C_VEL
LIN {X 0,Y 487.892,Z 898.656,A -85,B 0,C 180,E1 -6388.349,E2 -6388.349} C_VEL
LIN {X 0,Y 487.86,Z 895.316,A -85,B 0,C 180,E1 -6390,E2 -6390} C_VEL
LIN {X 0,Y 488.082,Z 891.874,A -85,B 0,C 180,E1 -6391.238,E2 -6391.238} C_VEL
LIN {X 0,Y 488.104,Z 887.523,A -85,B 0,C 180,E1 -6392.476,E2 -6392.476} C_VEL
LIN {X 0,Y 488.403,Z 882.221,A -85,B 0,C 180,E1 -6393.713,E2 -6393.713} C_VEL
LIN {X 0,Y 488.783,Z 874.641,A -85,B 0,C 180,E1 -6395.156,E2 -6395.156} C_VEL
LIN {X 0,Y 489.138,Z 866.758,A -85,B 0,C 180,E1 -6396.393,E2 -6396.393} C_VEL
LIN {X 0,Y 489.563,Z 856.579,A -85,B 0,C 180,E1 -6397.714,E2 -6397.714} C_VEL
LIN {X 0,Y 490.144,Z 845.722,A -85,B 0,C 180,E1 -6398.867,E2 -6398.867} C_VEL
LIN {X 0,Y 490.758,Z 833.893,A -85,B 0,C 180,E1 -6399.895,E2 -6399.895} C_VEL
LIN {X 0,Y 491.175,Z 822.282,A -85,B 0,C 180,E1 -6400.72,E2 -6400.72} C_VEL
LIN {X 0,Y 491.773,Z 809.57,A -85,B 0,C 180,E1 -6401.437,E2 -6401.437} C_VEL
LIN {X 0,Y 492.149,Z 796.605,A -85,B 0,C 180,E1 -6402.003,E2 -6402.003} C_VEL
LIN {X 0,Y 492.454,Z 782.608,A -85,B 0,C 180,E1 -6402.44,E2 -6402.44} C_VEL
LIN {X 0,Y 492.632,Z 766.206,A -85,B 0,C 180,E1 -6402.749,E2 -6402.749} C_VEL
LIN {X 0,Y 493.572,Z 656.432,A -85,B 0,C 180,E1 -6404.367,E2 -6404.367} C_VEL
LIN {X 0,Y 490.255,Z 640.501,A -85,B 0,C 180,E1 -6404.768,E2 -6404.768} C_VEL
LIN {X 0,Y 490.446,Z 632.592,A -85,B 0,C 180,E1 -6406.238,E2 -6406.238} C_VEL
LIN {X 0,Y 488.749,Z 623.732,A -85,B 0,C 180,E1 -6408.047,E2 -6408.047} C_VEL
LIN {X 0,Y 488.711,Z 623.736,A -85,B 0,C 180,E1 -6411.071,E2 -6411.071} C_VEL
LIN {X 0,Y 488.666,Z 623.737,A -85,B 0,C 180,E1 -6413.747,E2 -6413.747} C_VEL
LIN {X 0,Y 488.67,Z 623.741,A -85,B 0,C 180,E1 -6416.477,E2 -6416.477} C_VEL
LIN {X 0,Y 488.692,Z 623.735,A -85,B 0,C 180,E1 -6419.273,E2 -6419.273} C_VEL
LIN {X 0,Y 488.682,Z 623.735,A -85,B 0,C 180,E1 -6422.149,E2 -6422.149} C_VEL
LIN {X 0,Y 488.708,Z 623.735,A -85,B 0,C 180,E1 -6425.116,E2 -6425.116} C_VEL
LIN {X 0,Y 488.658,Z 623.737,A -85,B 0,C 180,E1 -6428.202,E2 -6428.202} C_VEL
LIN {X 0,Y 488.697,Z 623.725,A -85,B 0,C 180,E1 -6430.341,E2 -6430.341} C_VEL
LIN {X 0,Y 488.676,Z 623.733,A -85,B 0,C 180,E1 -6433.656,E2 -6433.656} C_VEL
LIN {X 0,Y 488.676,Z 623.734,A -85,B 0,C 180,E1 -6436.344,E2 -6436.344} C_VEL
LIN {X 0,Y 488.707,Z 623.731,A -85,B 0,C 180,E1 -6439.673,E2 -6439.673} C_VEL
LIN {X 0,Y 488.663,Z 623.73,A -85,B 0,C 180,E1 -6442.839,E2 -6442.839} C_VEL
LIN {X 0,Y 488.725,Z 623.728,A -85,B 0,C 180,E1 -6445.886,E2 -6445.886} C_VEL
LIN {X 0,Y 488.694,Z 623.733,A -85,B 0,C 180,E1 -6448.82,E2 -6448.82} C_VEL
LIN {X 0,Y 488.709,Z 623.733,A -85,B 0,C 180,E1 -6451.669,E2 -6451.669} C_VEL
LIN {X 0,Y 488.701,Z 623.732,A -85,B 0,C 180,E1 -6454.959,E2 -6454.959} C_VEL
LIN {X 0,Y 488.701,Z 623.731,A -85,B 0,C 180,E1 -6458.043,E2 -6458.043} C_VEL
LIN {X 0,Y 488.745,Z 623.724,A -85,B 0,C 180,E1 -6460.686,E2 -6460.686} C_VEL
LIN {X 0,Y 488.764,Z 623.722,A -85,B 0,C 180,E1 -6464.145,E2 -6464.145} C_VEL
LIN {X 0,Y 488.731,Z 623.727,A -85,B 0,C 180,E1 -6466.698,E2 -6466.698} C_VEL
LIN {X 0,Y 488.737,Z 623.725,A -85,B 0,C 180,E1 -6469.226,E2 -6469.226} C_VEL
LIN {X 0,Y 488.789,Z 623.726,A -85,B 0,C 180,E1 -6471.733,E2 -6471.733} C_VEL
LIN {X 0,Y 488.833,Z 623.715,A -85,B 0,C 180,E1 -6474.224,E2 -6474.224} C_VEL
LIN {X 0,Y 488.957,Z 623.702,A -85,B 0,C 180,E1 -6477.528,E2 -6477.528} C_VEL
LIN {X 0,Y 488.917,Z 623.7,A -85,B 0,C 180,E1 -6480.823,E2 -6480.823} C_VEL
LIN {X 0,Y 488.963,Z 623.699,A -85,B 0,C 180,E1 -6482.471,E2 -6482.471} C_VEL
LIN {X 0,Y 488.843,Z 623.718,A -85,B 0,C 180,E1 -6485.776,E2 -6485.776} C_VEL
LIN {X 0,Y 488.819,Z 623.72,A -85,B 0,C 180,E1 -6488.266,E2 -6488.266} C_VEL
LIN {X 0,Y 488.809,Z 623.717,A -85,B 0,C 180,E1 -6491.612,E2 -6491.612} C_VEL
LIN {X 0,Y 488.765,Z 623.72,A -85,B 0,C 180,E1 -6495,E2 -6495} C_VEL
LIN {X 0,Y 488.758,Z 623.725,A -85,B 0,C 180,E1 -6498.442,E2 -6498.442} C_VEL
LIN {X 0,Y 488.709,Z 623.728,A -85,B 0,C 180,E1 -6501.07,E2 -6501.07} C_VEL
LIN {X 0,Y 488.682,Z 623.733,A -85,B 0,C 180,E1 -6503.746,E2 -6503.746} C_VEL
LIN {X 0,Y 488.794,Z 623.717,A -85,B 0,C 180,E1 -6506.943,E2 -6506.943} C_VEL
LIN {X 0,Y 488.712,Z 623.735,A -85,B 0,C 180,E1 -6510.363,E2 -6510.363} C_VEL
LIN {X 0,Y 488.737,Z 623.726,A -85,B 0,C 180,E1 -6513.484,E2 -6513.484} C_VEL
LIN {X 0,Y 488.684,Z 623.74,A -85,B 0,C 180,E1 -6516.354,E2 -6516.354} C_VEL
LIN {X 0,Y 488.745,Z 623.724,A -85,B 0,C 180,E1 -6519.25,E2 -6519.25} C_VEL
LIN {X 0,Y 488.713,Z 623.729,A -85,B 0,C 180,E1 -6521.6,E2 -6521.6} C_VEL
LIN {X 0,Y 488.714,Z 623.734,A -85,B 0,C 180,E1 -6524.801,E2 -6524.801} C_VEL
LIN {X 0,Y 488.697,Z 623.73,A -85,B 0,C 180,E1 -6527.475,E2 -6527.475} C_VEL
LIN {X 0,Y 488.734,Z 623.727,A -85,B 0,C 180,E1 -6529.676,E2 -6529.676} C_VEL
LIN {X 0,Y 488.686,Z 623.74,A -85,B 0,C 180,E1 -6532.841,E2 -6532.841} C_VEL
LIN {X 0,Y 488.737,Z 623.728,A -85,B 0,C 180,E1 -6535.887,E2 -6535.887} C_VEL
LIN {X 0,Y 488.696,Z 623.733,A -85,B 0,C 180,E1 -6538.82,E2 -6538.82} C_VEL
LIN {X 0,Y 488.753,Z 623.729,A -85,B 0,C 180,E1 -6542.139,E2 -6542.139} C_VEL
LIN {X 0,Y 488.771,Z 623.732,A -85,B 0,C 180,E1 -6542.372,E2 -6542.372} C_VEL
LIN {X 0,Y 491.704,Z 637.12,A -85,B 0,C 180,E1 -6544.609,E2 -6544.609} C_VEL
LIN {X 0,Y 491.628,Z 644.408,A -85,B 0,C 180,E1 -6545.725,E2 -6545.725} C_VEL
LIN {X 0,Y 490.739,Z 665.199,A -85,B 0,C 180,E1 -6548.847,E2 -6548.847} C_VEL
LIN {X 0,Y 490.374,Z 674.793,A -85,B 0,C 180,E1 -6550.274,E2 -6550.274} C_VEL
LIN {X 0,Y 493.53,Z 692.951,A -85,B 0,C 180,E1 -6550.685,E2 -6550.685} C_VEL
LIN {X 0,Y 492.48,Z 813.47,A -85,B 0,C 180,E1 -6552.481,E2 -6552.481} C_VEL
LIN {X 0,Y 492.122,Z 828.02,A -85,B 0,C 180,E1 -6552.87,E2 -6552.87} C_VEL
LIN {X 0,Y 491.747,Z 841.383,A -85,B 0,C 180,E1 -6553.391,E2 -6553.391} C_VEL
LIN {X 0,Y 491.255,Z 853.598,A -85,B 0,C 180,E1 -6554.014,E2 -6554.014} C_VEL
LIN {X 0,Y 490.694,Z 866.456,A -85,B 0,C 180,E1 -6554.847,E2 -6554.847} C_VEL
LIN {X 0,Y 490.104,Z 878.151,A -85,B 0,C 180,E1 -6555.784,E2 -6555.784} C_VEL
LIN {X 0,Y 489.547,Z 889.852,A -85,B 0,C 180,E1 -6556.932,E2 -6556.932} C_VEL
LIN {X 0,Y 489.153,Z 899.282,A -85,B 0,C 180,E1 -6558.052,E2 -6558.052} C_VEL
LIN {X 0,Y 488.747,Z 907.602,A -85,B 0,C 180,E1 -6559.226,E2 -6559.226} C_VEL
LIN {X 0,Y 488.416,Z 916.152,A -85,B 0,C 180,E1 -6560.684,E2 -6560.684} C_VEL
LIN {X 0,Y 488.161,Z 923.044,A -85,B 0,C 180,E1 -6562.139,E2 -6562.139} C_VEL
LIN {X 0,Y 488.074,Z 928.181,A -85,B 0,C 180,E1 -6563.495,E2 -6563.495} C_VEL
LIN {X 0,Y 487.962,Z 932.724,A -85,B 0,C 180,E1 -6565.042,E2 -6565.042} C_VEL
LIN {X 0,Y 487.955,Z 936.15,A -85,B 0,C 180,E1 -6566.697,E2 -6566.697} C_VEL
LIN {X 0,Y 487.885,Z 938.174,A -85,B 0,C 180,E1 -6568.349,E2 -6568.349} C_VEL
LIN {X 0,Y 487.817,Z 938.843,A -85,B 0,C 180,E1 -6570,E2 -6570} C_VEL
LIN {X 0,Y 487.885,Z 938.174,A -85,B 0,C 180,E1 -6571.651,E2 -6571.651} C_VEL
LIN {X 0,Y 487.955,Z 936.15,A -85,B 0,C 180,E1 -6573.303,E2 -6573.303} C_VEL
LIN {X 0,Y 487.962,Z 932.72,A -85,B 0,C 180,E1 -6574.957,E2 -6574.957} C_VEL
LIN {X 0,Y 488.045,Z 928.274,A -85,B 0,C 180,E1 -6576.475,E2 -6576.475} C_VEL
LIN {X 0,Y 488.161,Z 923.031,A -85,B 0,C 180,E1 -6577.861,E2 -6577.861} C_VEL
LIN {X 0,Y 488.416,Z 916.139,A -85,B 0,C 180,E1 -6579.316,E2 -6579.316} C_VEL
LIN {X 0,Y 488.74,Z 907.585,A -85,B 0,C 180,E1 -6580.774,E2 -6580.774} C_VEL
LIN {X 0,Y 489.129,Z 899.281,A -85,B 0,C 180,E1 -6581.946,E2 -6581.946} C_VEL
LIN {X 0,Y 489.541,Z 889.829,A -85,B 0,C 180,E1 -6583.068,E2 -6583.068} C_VEL
LIN {X 0,Y 490.103,Z 878.124,A -85,B 0,C 180,E1 -6584.215,E2 -6584.215} C_VEL
LIN {X 0,Y 490.692,Z 866.431,A -85,B 0,C 180,E1 -6585.152,E2 -6585.152} C_VEL
LIN {X 0,Y 491.243,Z 853.566,A -85,B 0,C 180,E1 -6585.986,E2 -6585.986} C_VEL
LIN {X 0,Y 491.754,Z 840.32,A -85,B 0,C 180,E1 -6586.657,E2 -6586.657} C_VEL
LIN {X 0,Y 492.145,Z 826.359,A -85,B 0,C 180,E1 -6587.186,E2 -6587.186} C_VEL
LIN {X 0,Y 492.535,Z 812.165,A -85,B 0,C 180,E1 -6587.544,E2 -6587.544} C_VEL
LIN {X 0,Y 493.421,Z 692.17,A -85,B 0,C 180,E1 -6589.33,E2 -6589.33} C_VEL
LIN {X 0,Y 490.374,Z 674.754,A -85,B 0,C 180,E1 -6589.726,E2 -6589.726} C_VEL
LIN {X 0,Y 491.145,Z 654.645,A -85,B 0,C 180,E1 -6592.728,E2 -6592.728} C_VEL
LIN {X 0,Y 491.772,Z 640.084,A -85,B 0,C 180,E1 -6594.935,E2 -6594.935} C_VEL
LIN {X 0,Y 491.683,Z 637.169,A -85,B 0,C 180,E1 -6595.392,E2 -6595.392} C_VEL
LIN {X 0,Y 488.768,Z 623.729,A -85,B 0,C 180,E1 -6597.686,E2 -6597.686} C_VEL
LIN {X 0,Y 488.711,Z 623.732,A -85,B 0,C 180,E1 -6600.363,E2 -6600.363} C_VEL
LIN {X 0,Y 488.737,Z 623.729,A -85,B 0,C 180,E1 -6603.485,E2 -6603.485} C_VEL
LIN {X 0,Y 488.691,Z 623.731,A -85,B 0,C 180,E1 -6606.356,E2 -6606.356} C_VEL
LIN {X 0,Y 488.731,Z 623.734,A -85,B 0,C 180,E1 -6609.251,E2 -6609.251} C_VEL
LIN {X 0,Y 488.696,Z 623.732,A -85,B 0,C 180,E1 -6612.525,E2 -6612.525} C_VEL
LIN {X 0,Y 488.713,Z 623.732,A -85,B 0,C 180,E1 -6615.199,E2 -6615.199} C_VEL
LIN {X 0,Y 488.713,Z 623.726,A -85,B 0,C 180,E1 -6618.4,E2 -6618.4} C_VEL
LIN {X 0,Y 488.742,Z 623.727,A -85,B 0,C 180,E1 -6620.942,E2 -6620.942} C_VEL
LIN {X 0,Y 488.687,Z 623.737,A -85,B 0,C 180,E1 -6623.869,E2 -6623.869} C_VEL
LIN {X 0,Y 488.74,Z 623.724,A -85,B 0,C 180,E1 -6626.877,E2 -6626.877} C_VEL
LIN {X 0,Y 488.725,Z 623.726,A -85,B 0,C 180,E1 -6629.781,E2 -6629.781} C_VEL
LIN {X 0,Y 488.793,Z 623.718,A -85,B 0,C 180,E1 -6633.056,E2 -6633.056} C_VEL
LIN {X 0,Y 488.696,Z 623.733,A -85,B 0,C 180,E1 -6636.255,E2 -6636.255} C_VEL
LIN {X 0,Y 488.747,Z 623.725,A -85,B 0,C 180,E1 -6639.176,E2 -6639.176} C_VEL
LIN {X 0,Y 488.761,Z 623.725,A -85,B 0,C 180,E1 -6641.628,E2 -6641.628} C_VEL
LIN {X 0,Y 488.764,Z 623.722,A -85,B 0,C 180,E1 -6645,E2 -6645} C_VEL
LIN {X 0,Y 488.808,Z 623.722,A -85,B 0,C 180,E1 -6648.388,E2 -6648.388} C_VEL
LIN {X 0,Y 488.819,Z 623.715,A -85,B 0,C 180,E1 -6651.734,E2 -6651.734} C_VEL
LIN {X 0,Y 488.852,Z 623.718,A -85,B 0,C 180,E1 -6654.224,E2 -6654.224} C_VEL
LIN {X 0,Y 488.963,Z 623.698,A -85,B 0,C 180,E1 -6657.529,E2 -6657.529} C_VEL
LIN {X 0,Y 488.936,Z 623.701,A -85,B 0,C 180,E1 -6660.824,E2 -6660.824} C_VEL
LIN {X 0,Y 488.963,Z 623.706,A -85,B 0,C 180,E1 -6662.472,E2 -6662.472} C_VEL
LIN {X 0,Y 488.849,Z 623.709,A -85,B 0,C 180,E1 -6665.776,E2 -6665.776} C_VEL
LIN {X 0,Y 488.818,Z 623.722,A -85,B 0,C 180,E1 -6668.267,E2 -6668.267} C_VEL
LIN {X 0,Y 488.808,Z 623.716,A -85,B 0,C 180,E1 -6671.613,E2 -6671.613} C_VEL
LIN {X 0,Y 488.767,Z 623.723,A -85,B 0,C 180,E1 -6675.001,E2 -6675.001} C_VEL
LIN {X 0,Y 488.749,Z 623.73,A -85,B 0,C 180,E1 -6678.443,E2 -6678.443} C_VEL
LIN {X 0,Y 488.709,Z 623.734,A -85,B 0,C 180,E1 -6681.071,E2 -6681.071} C_VEL
LIN {X 0,Y 488.689,Z 623.729,A -85,B 0,C 180,E1 -6683.746,E2 -6683.746} C_VEL
LIN {X 0,Y 488.721,Z 623.732,A -85,B 0,C 180,E1 -6686.474,E2 -6686.474} C_VEL
LIN {X 0,Y 488.712,Z 623.724,A -85,B 0,C 180,E1 -6689.271,E2 -6689.271} C_VEL
LIN {X 0,Y 488.705,Z 623.731,A -85,B 0,C 180,E1 -6692.147,E2 -6692.147} C_VEL
LIN {X 0,Y 488.717,Z 623.736,A -85,B 0,C 180,E1 -6695.116,E2 -6695.116} C_VEL
LIN {X 0,Y 488.679,Z 623.734,A -85,B 0,C 180,E1 -6698.201,E2 -6698.201} C_VEL
LIN {X 0,Y 488.695,Z 623.729,A -85,B 0,C 180,E1 -6700.341,E2 -6700.341} C_VEL
LIN {X 0,Y 488.677,Z 623.737,A -85,B 0,C 180,E1 -6703.656,E2 -6703.656} C_VEL
LIN {X 0,Y 488.676,Z 623.734,A -85,B 0,C 180,E1 -6706.344,E2 -6706.344} C_VEL
LIN {X 0,Y 488.706,Z 623.736,A -85,B 0,C 180,E1 -6709.674,E2 -6709.674} C_VEL
LIN {X 0,Y 488.681,Z 623.738,A -85,B 0,C 180,E1 -6712.841,E2 -6712.841} C_VEL
LIN {X 0,Y 488.721,Z 623.73,A -85,B 0,C 180,E1 -6715.886,E2 -6715.886} C_VEL
LIN {X 0,Y 488.689,Z 623.736,A -85,B 0,C 180,E1 -6718.82,E2 -6718.82} C_VEL
LIN {X 0,Y 488.732,Z 623.858,A -85,B 0,C 180,E1 -6722.079,E2 -6722.079} C_VEL
LIN {X 0,Y 489.684,Z 628.569,A -85,B 0,C 180,E1 -6723.036,E2 -6723.036} C_VEL
LIN {X 0,Y 489.354,Z 630.691,A -85,B 0,C 180,E1 -6723.422,E2 -6723.422} C_VEL
LIN {X 0,Y 486.916,Z 634.445,A -85,B 0,C 180,E1 -6724.005,E2 -6724.005} C_VEL
LIN {X 0,Y 484.163,Z 638.272,A -85,B 0,C 180,E1 -6724.588,E2 -6724.588} C_VEL
LIN {X 0,Y 483.386,Z 640.523,A -85,B 0,C 180,E1 -6724.975,E2 -6724.975} C_VEL
LIN {X 0,Y 483.43,Z 641.199,A -85,B 0,C 180,E1 -6725.055,E2 -6725.055} C_VEL
LIN {X 0,Y 486.886,Z 657.193,A -85,B 0,C 180,E1 -6725.453,E2 -6725.453} C_VEL
LIN {X 0,Y 485.931,Z 776.937,A -85,B 0,C 180,E1 -6727.267,E2 -6727.267} C_VEL
LIN {X 0,Y 485.589,Z 791.125,A -85,B 0,C 180,E1 -6727.643,E2 -6727.643} C_VEL
LIN {X 0,Y 485.108,Z 803.775,A -85,B 0,C 180,E1 -6728.125,E2 -6728.125} C_VEL
LIN {X 0,Y 484.648,Z 816.033,A -85,B 0,C 180,E1 -6728.744,E2 -6728.744} C_VEL
LIN {X 0,Y 484.044,Z 829.32,A -85,B 0,C 180,E1 -6729.607,E2 -6729.607} C_VEL
LIN {X 0,Y 483.552,Z 840.097,A -85,B 0,C 180,E1 -6730.471,E2 -6730.471} C_VEL
LIN {X 0,Y 482.958,Z 851.184,A -85,B 0,C 180,E1 -6731.548,E2 -6731.548} C_VEL
LIN {X 0,Y 482.468,Z 860.428,A -85,B 0,C 180,E1 -6732.625,E2 -6732.625} C_VEL
LIN {X 0,Y 482.005,Z 869.648,A -85,B 0,C 180,E1 -6733.917,E2 -6733.917} C_VEL
LIN {X 0,Y 481.621,Z 877.29,A -85,B 0,C 180,E1 -6735.205,E2 -6735.205} C_VEL
LIN {X 0,Y 481.306,Z 883.632,A -85,B 0,C 180,E1 -6736.489,E2 -6736.489} C_VEL
LIN {X 0,Y 481.104,Z 888.812,A -85,B 0,C 180,E1 -6737.771,E2 -6737.771} C_VEL
LIN {X 0,Y 480.96,Z 893.005,A -85,B 0,C 180,E1 -6739.049,E2 -6739.049} C_VEL
LIN {X 0,Y 480.849,Z 897.22,A -85,B 0,C 180,E1 -6740.748,E2 -6740.748} C_VEL
LIN {X 0,Y 480.836,Z 899.976,A -85,B 0,C 180,E1 -6742.441,E2 -6742.441} C_VEL
LIN {X 0,Y 480.814,Z 901.366,A -85,B 0,C 180,E1 -6744.127,E2 -6744.127} C_VEL
LIN {X 0,Y 480.767,Z 901.434,A -85,B 0,C 180,E1 -6745.809,E2 -6745.809} C_VEL
LIN {X 0,Y 480.859,Z 900.968,A -85,B 0,C 180,E1 -6746.649,E2 -6746.649} C_VEL
LIN {X 0,Y 480.823,Z 899.052,A -85,B 0,C 180,E1 -6748.325,E2 -6748.325} C_VEL
LIN {X 0,Y 480.781,Z 895.771,A -85,B 0,C 180,E1 -6750,E2 -6750} C_VEL
LIN {X 0,Y 481.013,Z 892.359,A -85,B 0,C 180,E1 -6751.256,E2 -6751.256} C_VEL
LIN {X 0,Y 481.256,Z 886.459,A -85,B 0,C 180,E1 -6752.93,E2 -6752.93} C_VEL
LIN {X 0,Y 481.532,Z 879.834,A -85,B 0,C 180,E1 -6754.395,E2 -6754.395} C_VEL
LIN {X 0,Y 481.846,Z 872.917,A -85,B 0,C 180,E1 -6755.65,E2 -6755.65} C_VEL
LIN {X 0,Y 482.258,Z 864.622,A -85,B 0,C 180,E1 -6756.905,E2 -6756.905} C_VEL
LIN {X 0,Y 482.734,Z 855.089,A -85,B 0,C 180,E1 -6758.109,E2 -6758.109} C_VEL
LIN {X 0,Y 483.409,Z 843.483,A -85,B 0,C 180,E1 -6759.308,E2 -6759.308} C_VEL
LIN {X 0,Y 483.943,Z 832.421,A -85,B 0,C 180,E1 -6760.248,E2 -6760.248} C_VEL
LIN {X 0,Y 484.492,Z 820.374,A -85,B 0,C 180,E1 -6761.082,E2 -6761.082} C_VEL
LIN {X 0,Y 485.068,Z 807.001,A -85,B 0,C 180,E1 -6761.809,E2 -6761.809} C_VEL
LIN {X 0,Y 485.455,Z 793.016,A -85,B 0,C 180,E1 -6762.383,E2 -6762.383} C_VEL
LIN {X 0,Y 485.732,Z 779.278,A -85,B 0,C 180,E1 -6762.774,E2 -6762.774} C_VEL
LIN {X 0,Y 486.003,Z 755.538,A -85,B 0,C 180,E1 -6763.165,E2 -6763.165} C_VEL
LIN {X 0,Y 486.836,Z 656.828,A -85,B 0,C 180,E1 -6764.644,E2 -6764.644} C_VEL
LIN {X 0,Y 483.361,Z 640.801,A -85,B 0,C 180,E1 -6765.051,E2 -6765.051} C_VEL
LIN {X 0,Y 483.467,Z 633.766,A -85,B 0,C 180,E1 -6766.377,E2 -6766.377} C_VEL
LIN {X 0,Y 481.709,Z 624.61,A -85,B 0,C 180,E1 -6768.233,E2 -6768.233} C_VEL
LIN {X 0,Y 481.649,Z 624.613,A -85,B 0,C 180,E1 -6771.395,E2 -6771.395} C_VEL
LIN {X 0,Y 481.645,Z 624.613,A -85,B 0,C 180,E1 -6774.115,E2 -6774.115} C_VEL
LIN {X 0,Y 481.645,Z 624.616,A -85,B 0,C 180,E1 -6777.114,E2 -6777.114} C_VEL
LIN {X 0,Y 481.655,Z 624.61,A -85,B 0,C 180,E1 -6779.743,E2 -6779.743} C_VEL
LIN {X 0,Y 481.637,Z 624.618,A -85,B 0,C 180,E1 -6782.677,E2 -6782.677} C_VEL
LIN {X 0,Y 481.652,Z 624.613,A -85,B 0,C 180,E1 -6785.202,E2 -6785.202} C_VEL
LIN {X 0,Y 481.657,Z 624.612,A -85,B 0,C 180,E1 -6788.861,E2 -6788.861} C_VEL
LIN {X 0,Y 481.624,Z 624.612,A -85,B 0,C 180,E1 -6791.908,E2 -6791.908} C_VEL
LIN {X 0,Y 481.657,Z 624.608,A -85,B 0,C 180,E1 -6794.458,E2 -6794.458} C_VEL
LIN {X 0,Y 481.618,Z 624.619,A -85,B 0,C 180,E1 -6796.855,E2 -6796.855} C_VEL
LIN {X 0,Y 481.658,Z 624.607,A -85,B 0,C 180,E1 -6800.057,E2 -6800.057} C_VEL
LIN {X 0,Y 481.621,Z 624.609,A -85,B 0,C 180,E1 -6803.378,E2 -6803.378} C_VEL
LIN {X 0,Y 481.673,Z 624.606,A -85,B 0,C 180,E1 -6806.327,E2 -6806.327} C_VEL
LIN {X 0,Y 481.652,Z 624.61,A -85,B 0,C 180,E1 -6809.418,E2 -6809.418} C_VEL
LIN {X 0,Y 481.659,Z 624.608,A -85,B 0,C 180,E1 -6812.165,E2 -6812.165} C_VEL
LIN {X 0,Y 481.675,Z 624.607,A -85,B 0,C 180,E1 -6814.967,E2 -6814.967} C_VEL
LIN {X 0,Y 481.652,Z 624.613,A -85,B 0,C 180,E1 -6817.705,E2 -6817.705} C_VEL
LIN {X 0,Y 481.708,Z 624.6,A -85,B 0,C 180,E1 -6820.393,E2 -6820.393} C_VEL
LIN {X 0,Y 481.681,Z 624.599,A -85,B 0,C 180,E1 -6823.033,E2 -6823.033} C_VEL
LIN {X 0,Y 481.692,Z 624.611,A -85,B 0,C 180,E1 -6825.638,E2 -6825.638} C_VEL
LIN {X 0,Y 481.754,Z 624.593,A -85,B 0,C 180,E1 -6828.215,E2 -6828.215} C_VEL
LIN {X 0,Y 481.744,Z 624.601,A -85,B 0,C 180,E1 -6831.611,E2 -6831.611} C_VEL
LIN {X 0,Y 481.792,Z 624.593,A -85,B 0,C 180,E1 -6834.139,E2 -6834.139} C_VEL
LIN {X 0,Y 481.923,Z 624.578,A -85,B 0,C 180,E1 -6837.492,E2 -6837.492} C_VEL
LIN {X 0,Y 481.944,Z 624.575,A -85,B 0,C 180,E1 -6840,E2 -6840} C_VEL
LIN {X 0,Y 481.93,Z 624.575,A -85,B 0,C 180,E1 -6842.507,E2 -6842.507} C_VEL
LIN {X 0,Y 481.802,Z 624.595,A -85,B 0,C 180,E1 -6845.86,E2 -6845.86} C_VEL
LIN {X 0,Y 481.764,Z 624.597,A -85,B 0,C 180,E1 -6848.388,E2 -6848.388} C_VEL
LIN {X 0,Y 481.754,Z 624.598,A -85,B 0,C 180,E1 -6851.785,E2 -6851.785} C_VEL
LIN {X 0,Y 481.746,Z 624.594,A -85,B 0,C 180,E1 -6855.224,E2 -6855.224} C_VEL
LIN {X 0,Y 481.715,Z 624.599,A -85,B 0,C 180,E1 -6858.721,E2 -6858.721} C_VEL
LIN {X 0,Y 481.648,Z 624.608,A -85,B 0,C 180,E1 -6861.394,E2 -6861.394} C_VEL
LIN {X 0,Y 481.663,Z 624.611,A -85,B 0,C 180,E1 -6864.114,E2 -6864.114} C_VEL
LIN {X 0,Y 481.749,Z 624.594,A -85,B 0,C 180,E1 -6867.139,E2 -6867.139} C_VEL
LIN {X 0,Y 481.681,Z 624.607,A -85,B 0,C 180,E1 -6869.741,E2 -6869.741} C_VEL
LIN {X 0,Y 481.674,Z 624.61,A -85,B 0,C 180,E1 -6872.674,E2 -6872.674} C_VEL
LIN {X 0,Y 481.639,Z 624.612,A -85,B 0,C 180,E1 -6875.709,E2 -6875.709} C_VEL
LIN {X 0,Y 481.716,Z 624.599,A -85,B 0,C 180,E1 -6879.354,E2 -6879.354} C_VEL
LIN {X 0,Y 481.65,Z 624.613,A -85,B 0,C 180,E1 -6882.16,E2 -6882.16} C_VEL
LIN {X 0,Y 481.662,Z 624.607,A -85,B 0,C 180,E1 -6885.543,E2 -6885.543} C_VEL
LIN {X 0,Y 481.664,Z 624.608,A -85,B 0,C 180,E1 -6888.086,E2 -6888.086} C_VEL
LIN {X 0,Y 481.673,Z 624.609,A -85,B 0,C 180,E1 -6891.141,E2 -6891.141} C_VEL
LIN {X 0,Y 481.671,Z 624.614,A -85,B 0,C 180,E1 -6894.794,E2 -6894.794} C_VEL
LIN {X 0,Y 481.675,Z 624.609,A -85,B 0,C 180,E1 -6897.326,E2 -6897.326} C_VEL
LIN {X 0,Y 481.681,Z 624.611,A -85,B 0,C 180,E1 -6900.259,E2 -6900.259} C_VEL
LIN {X 0,Y 481.727,Z 624.656,A -85,B 0,C 180,E1 -6902.14,E2 -6902.14} C_VEL
LIN {X 0,Y 484.711,Z 638.264,A -85,B 0,C 180,E1 -6904.446,E2 -6904.446} C_VEL
LIN {X 0,Y 484.894,Z 642.684,A -85,B 0,C 180,E1 -6905.145,E2 -6905.145} C_VEL
LIN {X 0,Y 483.879,Z 664.65,A -85,B 0,C 180,E1 -6908.489,E2 -6908.489} C_VEL
LIN {X 0,Y 483.441,Z 674.529,A -85,B 0,C 180,E1 -6909.979,E2 -6909.979} C_VEL
LIN {X 0,Y 486.83,Z 693.83,A -85,B 0,C 180,E1 -6910.426,E2 -6910.426} C_VEL
LIN {X 0,Y 485.707,Z 813.188,A -85,B 0,C 180,E1 -6912.229,E2 -6912.229} C_VEL
LIN {X 0,Y 485.334,Z 827.742,A -85,B 0,C 180,E1 -6912.623,E2 -6912.623} C_VEL
LIN {X 0,Y 484.923,Z 841.106,A -85,B 0,C 180,E1 -6913.15,E2 -6913.15} C_VEL
LIN {X 0,Y 484.379,Z 853.419,A -85,B 0,C 180,E1 -6913.787,E2 -6913.787} C_VEL
LIN {X 0,Y 483.795,Z 866.18,A -85,B 0,C 180,E1 -6914.626,E2 -6914.626} C_VEL
LIN {X 0,Y 483.184,Z 877.876,A -85,B 0,C 180,E1 -6915.576,E2 -6915.576} C_VEL
LIN {X 0,Y 482.57,Z 889.577,A -85,B 0,C 180,E1 -6916.739,E2 -6916.739} C_VEL
LIN {X 0,Y 482.071,Z 900.512,A -85,B 0,C 180,E1 -6918.071,E2 -6918.071} C_VEL
LIN {X 0,Y 481.594,Z 909.967,A -85,B 0,C 180,E1 -6919.489,E2 -6919.489} C_VEL
LIN {X 0,Y 481.276,Z 917.99,A -85,B 0,C 180,E1 -6920.968,E2 -6920.968} C_VEL
LIN {X 0,Y 481.013,Z 924.451,A -85,B 0,C 180,E1 -6922.444,E2 -6922.444} C_VEL
LIN {X 0,Y 480.934,Z 930.185,A -85,B 0,C 180,E1 -6924.129,E2 -6924.129} C_VEL
LIN {X 0,Y 480.815,Z 934.342,A -85,B 0,C 180,E1 -6925.809,E2 -6925.809} C_VEL
LIN {X 0,Y 480.879,Z 935.878,A -85,B 0,C 180,E1 -6926.649,E2 -6926.649} C_VEL
LIN {X 0,Y 480.815,Z 937.903,A -85,B 0,C 180,E1 -6928.325,E2 -6928.325} C_VEL
LIN {X 0,Y 480.741,Z 938.571,A -85,B 0,C 180,E1 -6930,E2 -6930} C_VEL
LIN {X 0,Y 480.815,Z 937.901,A -85,B 0,C 180,E1 -6931.675,E2 -6931.675} C_VEL
LIN {X 0,Y 480.879,Z 935.876,A -85,B 0,C 180,E1 -6933.351,E2 -6933.351} C_VEL
LIN {X 0,Y 480.894,Z 932.446,A -85,B 0,C 180,E1 -6935.03,E2 -6935.03} C_VEL
LIN {X 0,Y 480.961,Z 927.51,A -85,B 0,C 180,E1 -6936.713,E2 -6936.713} C_VEL
LIN {X 0,Y 481.169,Z 920.929,A -85,B 0,C 180,E1 -6938.399,E2 -6938.399} C_VEL
LIN {X 0,Y 481.432,Z 913.608,A -85,B 0,C 180,E1 -6939.877,E2 -6939.877} C_VEL
LIN {X 0,Y 481.906,Z 904.55,A -85,B 0,C 180,E1 -6941.355,E2 -6941.355} C_VEL
LIN {X 0,Y 482.327,Z 895.045,A -85,B 0,C 180,E1 -6942.625,E2 -6942.625} C_VEL
LIN {X 0,Y 482.804,Z 884.528,A -85,B 0,C 180,E1 -6943.79,E2 -6943.79} C_VEL
LIN {X 0,Y 483.402,Z 872.934,A -85,B 0,C 180,E1 -6944.847,E2 -6944.847} C_VEL
LIN {X 0,Y 484.093,Z 860.081,A -85,B 0,C 180,E1 -6945.796,E2 -6945.796} C_VEL
LIN {X 0,Y 484.61,Z 847.912,A -85,B 0,C 180,E1 -6946.515,E2 -6946.515} C_VEL
LIN {X 0,Y 485.11,Z 834.357,A -85,B 0,C 180,E1 -6947.136,E2 -6947.136} C_VEL
LIN {X 0,Y 485.544,Z 821.103,A -85,B 0,C 180,E1 -6947.576,E2 -6947.576} C_VEL
LIN {X 0,Y 485.802,Z 807.355,A -85,B 0,C 180,E1 -6947.877,E2 -6947.877} C_VEL
LIN {X 0,Y 486.742,Z 693.156,A -85,B 0,C 180,E1 -6949.587,E2 -6949.587} C_VEL
LIN {X 0,Y 483.452,Z 674.49,A -85,B 0,C 180,E1 -6950.02,E2 -6950.02} C_VEL
LIN {X 0,Y 484.251,Z 655.878,A -85,B 0,C 180,E1 -6952.844,E2 -6952.844} C_VEL
LIN {X 0,Y 484.915,Z 641.356,A -85,B 0,C 180,E1 -6955.083,E2 -6955.083} C_VEL
LIN {X 0,Y 484.42,Z 636.99,A -85,B 0,C 180,E1 -6955.801,E2 -6955.801} C_VEL
LIN {X 0,Y 481.712,Z 624.607,A -85,B 0,C 180,E1 -6957.979,E2 -6957.979} C_VEL
LIN {X 0,Y 481.648,Z 624.613,A -85,B 0,C 180,E1 -6960.711,E2 -6960.711} C_VEL
LIN {X 0,Y 481.697,Z 624.605,A -85,B 0,C 180,E1 -6963.733,E2 -6963.733} C_VEL
LIN {X 0,Y 481.632,Z 624.612,A -85,B 0,C 180,E1 -6966.746,E2 -6966.746} C_VEL
LIN {X 0,Y 481.686,Z 624.604,A -85,B 0,C 180,E1 -6969.94,E2 -6969.94} C_VEL
LIN {X 0,Y 481.667,Z 624.611,A -85,B 0,C 180,E1 -6973.297,E2 -6973.297} C_VEL
LIN {X 0,Y 481.659,Z 624.615,A -85,B 0,C 180,E1 -6975.641,E2 -6975.641} C_VEL
LIN {X 0,Y 481.669,Z 624.605,A -85,B 0,C 180,E1 -6978.96,E2 -6978.96} C_VEL
LIN {X 0,Y 481.699,Z 624.606,A -85,B 0,C 180,E1 -6981.144,E2 -6981.144} C_VEL
LIN {X 0,Y 481.67,Z 624.606,A -85,B 0,C 180,E1 -6984.795,E2 -6984.795} C_VEL
LIN {X 0,Y 481.674,Z 624.607,A -85,B 0,C 180,E1 -6987.326,E2 -6987.326} C_VEL
LIN {X 0,Y 481.68,Z 624.606,A -85,B 0,C 180,E1 -6990.259,E2 -6990.259} C_VEL
LIN {X 0,Y 481.747,Z 624.596,A -85,B 0,C 180,E1 -6993.112,E2 -6993.112} C_VEL
LIN {X 0,Y 481.679,Z 624.613,A -85,B 0,C 180,E1 -6995.887,E2 -6995.887} C_VEL
LIN {X 0,Y 481.704,Z 624.602,A -85,B 0,C 180,E1 -6999.028,E2 -6999.028} C_VEL
LIN {X 0,Y 481.71,Z 624.606,A -85,B 0,C 180,E1 -7002.159,E2 -7002.159} C_VEL
LIN {X 0,Y 481.744,Z 624.597,A -85,B 0,C 180,E1 -7004.776,E2 -7004.776} C_VEL
LIN {X 0,Y 481.753,Z 624.604,A -85,B 0,C 180,E1 -7008.215,E2 -7008.215} C_VEL
LIN {X 0,Y 481.764,Z 624.592,A -85,B 0,C 180,E1 -7011.612,E2 -7011.612} C_VEL
LIN {X 0,Y 481.812,Z 624.597,A -85,B 0,C 180,E1 -7014.14,E2 -7014.14} C_VEL
LIN {X 0,Y 481.93,Z 624.574,A -85,B 0,C 180,E1 -7017.493,E2 -7017.493} C_VEL
LIN {X 0,Y 481.887,Z 624.579,A -85,B 0,C 180,E1 -7020.836,E2 -7020.836} C_VEL
LIN {X 0,Y 481.929,Z 624.581,A -85,B 0,C 180,E1 -7022.508,E2 -7022.508} C_VEL
LIN {X 0,Y 481.81,Z 624.586,A -85,B 0,C 180,E1 -7025.861,E2 -7025.861} C_VEL
LIN {X 0,Y 481.764,Z 624.602,A -85,B 0,C 180,E1 -7028.389,E2 -7028.389} C_VEL
LIN {X 0,Y 481.753,Z 624.595,A -85,B 0,C 180,E1 -7031.785,E2 -7031.785} C_VEL
LIN {X 0,Y 481.747,Z 624.596,A -85,B 0,C 180,E1 -7035.224,E2 -7035.224} C_VEL
LIN {X 0,Y 481.711,Z 624.606,A -85,B 0,C 180,E1 -7038.722,E2 -7038.722} C_VEL
LIN {X 0,Y 481.648,Z 624.611,A -85,B 0,C 180,E1 -7041.395,E2 -7041.395} C_VEL
LIN {X 0,Y 481.673,Z 624.604,A -85,B 0,C 180,E1 -7044.114,E2 -7044.114} C_VEL
LIN {X 0,Y 481.697,Z 624.602,A -85,B 0,C 180,E1 -7047.127,E2 -7047.127} C_VEL
LIN {X 0,Y 481.675,Z 624.598,A -85,B 0,C 180,E1 -7049.742,E2 -7049.742} C_VEL
LIN {X 0,Y 481.673,Z 624.611,A -85,B 0,C 180,E1 -7052.675,E2 -7052.675} C_VEL
LIN {X 0,Y 481.638,Z 624.611,A -85,B 0,C 180,E1 -7055.71,E2 -7055.71} C_VEL
LIN {X 0,Y 481.668,Z 624.613,A -85,B 0,C 180,E1 -7058.86,E2 -7058.86} C_VEL
LIN {X 0,Y 481.629,Z 624.611,A -85,B 0,C 180,E1 -7062.163,E2 -7062.163} C_VEL
LIN {X 0,Y 481.656,Z 624.611,A -85,B 0,C 180,E1 -7065.542,E2 -7065.542} C_VEL
LIN {X 0,Y 481.626,Z 624.619,A -85,B 0,C 180,E1 -7068.955,E2 -7068.955} C_VEL
LIN {X 0,Y 481.655,Z 624.611,A -85,B 0,C 180,E1 -7071.993,E2 -7071.993} C_VEL
LIN {X 0,Y 481.685,Z 624.612,A -85,B 0,C 180,E1 -7075.318,E2 -7075.318} C_VEL
LIN {X 0,Y 481.642,Z 624.613,A -85,B 0,C 180,E1 -7078.311,E2 -7078.311} C_VEL
LIN {X 0,Y 481.663,Z 624.615,A -85,B 0,C 180,E1 -7081.216,E2 -7081.216} C_VEL
LIN {X 0,Y 481.665,Z 624.615,A -85,B 0,C 180,E1 -7081.811,E2 -7081.811} C_VEL
LIN {X 0,Y 483.589,Z 634.929,A -85,B 0,C 180,E1 -7083.92,E2 -7083.92} C_VEL
LIN {X 0,Y 483.386,Z 640.523,A -85,B 0,C 180,E1 -7084.975,E2 -7084.975} C_VEL
LIN {X 0,Y 482.932,Z 641.799,A -85,B 0,C 180,E1 -7085.043,E2 -7085.043} C_VEL
LIN {X 0,Y 477.437,Z 651.356,A -85,B 0,C 180,E1 -7084.943,E2 -7084.943} C_VEL
LIN {X 0,Y 476.431,Z 655.04,A -85,B 0,C 180,E1 -7084.945,E2 -7084.945} C_VEL
LIN {X 0,Y 476.773,Z 658.962,A -85,B 0,C 180,E1 -7084.986,E2 -7084.986} C_VEL
LIN {X 0,Y 479.98,Z 669.762,A -85,B 0,C 180,E1 -7085.343,E2 -7085.343} C_VEL
LIN {X 0,Y 480.147,Z 672.046,A -85,B 0,C 180,E1 -7085.391,E2 -7085.391} C_VEL
LIN {X 0,Y 479.188,Z 777.519,A -85,B 0,C 180,E1 -7087.015,E2 -7087.015} C_VEL
LIN {X 0,Y 478.84,Z 791.587,A -85,B 0,C 180,E1 -7087.396,E2 -7087.396} C_VEL
LIN {X 0,Y 478.312,Z 804.407,A -85,B 0,C 180,E1 -7087.894,E2 -7087.894} C_VEL
LIN {X 0,Y 477.811,Z 816.855,A -85,B 0,C 180,E1 -7088.538,E2 -7088.538} C_VEL
LIN {X 0,Y 477.249,Z 828.581,A -85,B 0,C 180,E1 -7089.303,E2 -7089.303} C_VEL
LIN {X 0,Y 476.669,Z 840.566,A -85,B 0,C 180,E1 -7090.274,E2 -7090.274} C_VEL
LIN {X 0,Y 476.102,Z 850.768,A -85,B 0,C 180,E1 -7091.273,E2 -7091.273} C_VEL
LIN {X 0,Y 475.456,Z 861.772,A -85,B 0,C 180,E1 -7092.583,E2 -7092.583} C_VEL
LIN {X 0,Y 474.986,Z 870.537,A -85,B 0,C 180,E1 -7093.849,E2 -7093.849} C_VEL
LIN {X 0,Y 474.574,Z 878.296,A -85,B 0,C 180,E1 -7095.199,E2 -7095.199} C_VEL
LIN {X 0,Y 474.216,Z 885.408,A -85,B 0,C 180,E1 -7096.72,E2 -7096.72} C_VEL
LIN {X 0,Y 473.985,Z 890.703,A -85,B 0,C 180,E1 -7098.132,E2 -7098.132} C_VEL
LIN {X 0,Y 473.882,Z 895.39,A -85,B 0,C 180,E1 -7099.749,E2 -7099.749} C_VEL
LIN {X 0,Y 473.747,Z 898.921,A -85,B 0,C 180,E1 -7101.469,E2 -7101.469} C_VEL
LIN {X 0,Y 473.788,Z 901.04,A -85,B 0,C 180,E1 -7103.185,E2 -7103.185} C_VEL
LIN {X 0,Y 473.738,Z 901.822,A -85,B 0,C 180,E1 -7104.893,E2 -7104.893} C_VEL
LIN {X 0,Y 473.783,Z 901.285,A -85,B 0,C 180,E1 -7106.598,E2 -7106.598} C_VEL
LIN {X 0,Y 473.755,Z 899.437,A -85,B 0,C 180,E1 -7108.3,E2 -7108.3} C_VEL
LIN {X 0,Y 473.705,Z 896.226,A -85,B 0,C 180,E1 -7110,E2 -7110} C_VEL
LIN {X 0,Y 473.948,Z 892.843,A -85,B 0,C 180,E1 -7111.275,E2 -7111.275} C_VEL
LIN {X 0,Y 473.987,Z 888.62,A -85,B 0,C 180,E1 -7112.55,E2 -7112.55} C_VEL
LIN {X 0,Y 474.311,Z 883.456,A -85,B 0,C 180,E1 -7113.823,E2 -7113.823} C_VEL
LIN {X 0,Y 474.743,Z 876.027,A -85,B 0,C 180,E1 -7115.309,E2 -7115.309} C_VEL
LIN {X 0,Y 475.125,Z 868.319,A -85,B 0,C 180,E1 -7116.583,E2 -7116.583} C_VEL
LIN {X 0,Y 475.492,Z 860.024,A -85,B 0,C 180,E1 -7117.736,E2 -7117.736} C_VEL
LIN {X 0,Y 476.15,Z 849.822,A -85,B 0,C 180,E1 -7118.916,E2 -7118.916} C_VEL
LIN {X 0,Y 476.83,Z 838.734,A -85,B 0,C 180,E1 -7119.973,E2 -7119.973} C_VEL
LIN {X 0,Y 477.387,Z 826.526,A -85,B 0,C 180,E1 -7120.926,E2 -7120.926} C_VEL
LIN {X 0,Y 477.998,Z 814.771,A -85,B 0,C 180,E1 -7121.664,E2 -7121.664} C_VEL
LIN {X 0,Y 478.483,Z 801.961,A -85,B 0,C 180,E1 -7122.297,E2 -7122.297} C_VEL
LIN {X 0,Y 478.852,Z 788.241,A -85,B 0,C 180,E1 -7122.799,E2 -7122.799} C_VEL
LIN {X 0,Y 479.112,Z 774.024,A -85,B 0,C 180,E1 -7123.142,E2 -7123.142} C_VEL
LIN {X 0,Y 480.138,Z 657.72,A -85,B 0,C 180,E1 -7124.916,E2 -7124.916} C_VEL
LIN {X 0,Y 476.467,Z 641.05,A -85,B 0,C 180,E1 -7125.348,E2 -7125.348} C_VEL
LIN {X 0,Y 476.506,Z 634.889,A -85,B 0,C 180,E1 -7126.525,E2 -7126.525} C_VEL
LIN {X 0,Y 474.671,Z 625.487,A -85,B 0,C 180,E1 -7128.478,E2 -7128.478} C_VEL
LIN {X 0,Y 474.639,Z 625.489,A -85,B 0,C 180,E1 -7131.116,E2 -7131.116} C_VEL
LIN {X 0,Y 474.623,Z 625.492,A -85,B 0,C 180,E1 -7134.495,E2 -7134.495} C_VEL
LIN {X 0,Y 474.596,Z 625.492,A -85,B 0,C 180,E1 -7137.327,E2 -7137.327} C_VEL
LIN {X 0,Y 474.583,Z 625.492,A -85,B 0,C 180,E1 -7140.232,E2 -7140.232} C_VEL
LIN {X 0,Y 474.611,Z 625.49,A -85,B 0,C 180,E1 -7143.223,E2 -7143.223} C_VEL
LIN {X 0,Y 474.575,Z 625.492,A -85,B 0,C 180,E1 -7146.325,E2 -7146.325} C_VEL
LIN {X 0,Y 474.603,Z 625.48,A -85,B 0,C 180,E1 -7149.643,E2 -7149.643} C_VEL
LIN {X 0,Y 474.572,Z 625.499,A -85,B 0,C 180,E1 -7152.939,E2 -7152.939} C_VEL
LIN {X 0,Y 474.604,Z 625.487,A -85,B 0,C 180,E1 -7155.894,E2 -7155.894} C_VEL
LIN {X 0,Y 474.594,Z 625.492,A -85,B 0,C 180,E1 -7159.339,E2 -7159.339} C_VEL
LIN {X 0,Y 474.595,Z 625.48,A -85,B 0,C 180,E1 -7161.707,E2 -7161.707} C_VEL
LIN {X 0,Y 474.621,Z 625.481,A -85,B 0,C 180,E1 -7164.725,E2 -7164.725} C_VEL
LIN {X 0,Y 474.638,Z 625.483,A -85,B 0,C 180,E1 -7167.787,E2 -7167.787} C_VEL
LIN {X 0,Y 474.609,Z 625.484,A -85,B 0,C 180,E1 -7170.888,E2 -7170.888} C_VEL
LIN {X 0,Y 474.586,Z 625.492,A -85,B 0,C 180,E1 -7173.624,E2 -7173.624} C_VEL
LIN {X 0,Y 474.637,Z 625.477,A -85,B 0,C 180,E1 -7176.642,E2 -7176.642} C_VEL
LIN {X 0,Y 474.657,Z 625.48,A -85,B 0,C 180,E1 -7180.089,E2 -7180.089} C_VEL
LIN {X 0,Y 474.641,Z 625.474,A -85,B 0,C 180,E1 -7182.774,E2 -7182.774} C_VEL
LIN {X 0,Y 474.65,Z 625.486,A -85,B 0,C 180,E1 -7185.421,E2 -7185.421} C_VEL
LIN {X 0,Y 474.708,Z 625.472,A -85,B 0,C 180,E1 -7188.037,E2 -7188.037} C_VEL
LIN {X 0,Y 474.715,Z 625.474,A -85,B 0,C 180,E1 -7191.486,E2 -7191.486} C_VEL
LIN {X 0,Y 474.745,Z 625.468,A -85,B 0,C 180,E1 -7194.904,E2 -7194.904} C_VEL
LIN {X 0,Y 474.889,Z 625.454,A -85,B 0,C 180,E1 -7197.455,E2 -7197.455} C_VEL
LIN {X 0,Y 474.914,Z 625.45,A -85,B 0,C 180,E1 -7200,E2 -7200} C_VEL
LIN {X 0,Y 474.896,Z 625.451,A -85,B 0,C 180,E1 -7202.544,E2 -7202.544} C_VEL
LIN {X 0,Y 474.763,Z 625.471,A -85,B 0,C 180,E1 -7205.948,E2 -7205.948} C_VEL
LIN {X 0,Y 474.729,Z 625.472,A -85,B 0,C 180,E1 -7208.513,E2 -7208.513} C_VEL
LIN {X 0,Y 474.707,Z 625.479,A -85,B 0,C 180,E1 -7211.962,E2 -7211.962} C_VEL
LIN {X 0,Y 474.705,Z 625.476,A -85,B 0,C 180,E1 -7215.777,E2 -7215.777} C_VEL
LIN {X 0,Y 474.668,Z 625.476,A -85,B 0,C 180,E1 -7219.01,E2 -7219.01} C_VEL
LIN {X 0,Y 474.591,Z 625.49,A -85,B 0,C 180,E1 -7221.729,E2 -7221.729} C_VEL
LIN {X 0,Y 474.643,Z 625.486,A -85,B 0,C 180,E1 -7224.494,E2 -7224.494} C_VEL
LIN {X 0,Y 474.683,Z 625.474,A -85,B 0,C 180,E1 -7227.334,E2 -7227.334} C_VEL
LIN {X 0,Y 474.608,Z 625.493,A -85,B 0,C 180,E1 -7230.23,E2 -7230.23} C_VEL
LIN {X 0,Y 474.645,Z 625.481,A -85,B 0,C 180,E1 -7233.22,E2 -7233.22} C_VEL
LIN {X 0,Y 474.591,Z 625.496,A -85,B 0,C 180,E1 -7236.323,E2 -7236.323} C_VEL
LIN {X 0,Y 474.653,Z 625.48,A -85,B 0,C 180,E1 -7239.651,E2 -7239.651} C_VEL
LIN {X 0,Y 474.617,Z 625.488,A -85,B 0,C 180,E1 -7242.934,E2 -7242.934} C_VEL
LIN {X 0,Y 474.617,Z 625.486,A -85,B 0,C 180,E1 -7245.896,E2 -7245.896} C_VEL
LIN {X 0,Y 474.634,Z 625.487,A -85,B 0,C 180,E1 -7249.04,E2 -7249.04} C_VEL
LIN {X 0,Y 474.613,Z 625.487,A -85,B 0,C 180,E1 -7251.704,E2 -7251.704} C_VEL
LIN {X 0,Y 474.632,Z 625.491,A -85,B 0,C 180,E1 -7254.726,E2 -7254.726} C_VEL
LIN {X 0,Y 474.639,Z 625.484,A -85,B 0,C 180,E1 -7257.788,E2 -7257.788} C_VEL
LIN {X 0,Y 474.626,Z 625.491,A -85,B 0,C 180,E1 -7260.884,E2 -7260.884} C_VEL
LIN {X 0,Y 474.668,Z 625.484,A -85,B 0,C 180,E1 -7261.884,E2 -7261.884} C_VEL
LIN {X 0,Y 477.78,Z 639.633,A -85,B 0,C 180,E1 -7264.321,E2 -7264.321} C_VEL
LIN {X 0,Y 478.021,Z 643.817,A -85,B 0,C 180,E1 -7264.995,E2 -7264.995} C_VEL
LIN {X 0,Y 476.934,Z 665.774,A -85,B 0,C 180,E1 -7268.383,E2 -7268.383} C_VEL
LIN {X 0,Y 476.547,Z 674.233,A -85,B 0,C 180,E1 -7269.677,E2 -7269.677} C_VEL
LIN {X 0,Y 480.085,Z 694.358,A -85,B 0,C 180,E1 -7270.153,E2 -7270.153} C_VEL
LIN {X 0,Y 478.989,Z 811.627,A -85,B 0,C 180,E1 -7271.943,E2 -7271.943} C_VEL
LIN {X 0,Y 478.594,Z 825.932,A -85,B 0,C 180,E1 -7272.315,E2 -7272.315} C_VEL
LIN {X 0,Y 478.156,Z 839.079,A -85,B 0,C 180,E1 -7272.819,E2 -7272.819} C_VEL
LIN {X 0,Y 477.619,Z 851.76,A -85,B 0,C 180,E1 -7273.465,E2 -7273.465} C_VEL
LIN {X 0,Y 477.017,Z 864.474,A -85,B 0,C 180,E1 -7274.293,E2 -7274.293} C_VEL
LIN {X 0,Y 476.34,Z 876.421,A -85,B 0,C 180,E1 -7275.255,E2 -7275.255} C_VEL
LIN {X 0,Y 475.732,Z 887.341,A -85,B 0,C 180,E1 -7276.328,E2 -7276.328} C_VEL
LIN {X 0,Y 475.171,Z 898.215,A -85,B 0,C 180,E1 -7277.626,E2 -7277.626} C_VEL
LIN {X 0,Y 474.727,Z 907.055,A -85,B 0,C 180,E1 -7278.904,E2 -7278.904} C_VEL
LIN {X 0,Y 474.353,Z 914.479,A -85,B 0,C 180,E1 -7280.19,E2 -7280.19} C_VEL
LIN {X 0,Y 474.102,Z 920.672,A -85,B 0,C 180,E1 -7281.475,E2 -7281.475} C_VEL
LIN {X 0,Y 473.896,Z 927.252,A -85,B 0,C 180,E1 -7283.186,E2 -7283.186} C_VEL
LIN {X 0,Y 473.825,Z 932.179,A -85,B 0,C 180,E1 -7284.894,E2 -7284.894} C_VEL
LIN {X 0,Y 473.786,Z 935.606,A -85,B 0,C 180,E1 -7286.598,E2 -7286.598} C_VEL
LIN {X 0,Y 473.718,Z 937.63,A -85,B 0,C 180,E1 -7288.3,E2 -7288.3} C_VEL
LIN {X 0,Y 473.667,Z 938.299,A -85,B 0,C 180,E1 -7290,E2 -7290} C_VEL
LIN {X 0,Y 473.718,Z 937.628,A -85,B 0,C 180,E1 -7291.7,E2 -7291.7} C_VEL
LIN {X 0,Y 473.786,Z 935.602,A -85,B 0,C 180,E1 -7293.402,E2 -7293.402} C_VEL
LIN {X 0,Y 473.825,Z 932.171,A -85,B 0,C 180,E1 -7295.106,E2 -7295.106} C_VEL
LIN {X 0,Y 473.891,Z 927.234,A -85,B 0,C 180,E1 -7296.814,E2 -7296.814} C_VEL
LIN {X 0,Y 474.101,Z 920.651,A -85,B 0,C 180,E1 -7298.525,E2 -7298.525} C_VEL
LIN {X 0,Y 474.381,Z 913.328,A -85,B 0,C 180,E1 -7300.025,E2 -7300.025} C_VEL
LIN {X 0,Y 474.881,Z 904.269,A -85,B 0,C 180,E1 -7301.525,E2 -7301.525} C_VEL
LIN {X 0,Y 475.325,Z 894.763,A -85,B 0,C 180,E1 -7302.814,E2 -7302.814} C_VEL
LIN {X 0,Y 475.841,Z 884.246,A -85,B 0,C 180,E1 -7303.996,E2 -7303.996} C_VEL
LIN {X 0,Y 476.498,Z 872.651,A -85,B 0,C 180,E1 -7305.067,E2 -7305.067} C_VEL
LIN {X 0,Y 477.236,Z 859.798,A -85,B 0,C 180,E1 -7306.029,E2 -7306.029} C_VEL
LIN {X 0,Y 477.842,Z 846.49,A -85,B 0,C 180,E1 -7306.818,E2 -7306.818} C_VEL
LIN {X 0,Y 478.393,Z 832.898,A -85,B 0,C 180,E1 -7307.434,E2 -7307.434} C_VEL
LIN {X 0,Y 478.829,Z 818.766,A -85,B 0,C 180,E1 -7307.892,E2 -7307.892} C_VEL
LIN {X 0,Y 479.104,Z 803.764,A -85,B 0,C 180,E1 -7308.19,E2 -7308.19} C_VEL
LIN {X 0,Y 479.98,Z 693.686,A -85,B 0,C 180,E1 -7309.863,E2 -7309.863} C_VEL
LIN {X 0,Y 476.54,Z 674.243,A -85,B 0,C 180,E1 -7310.323,E2 -7310.323} C_VEL
LIN {X 0,Y 477.38,Z 655.689,A -85,B 0,C 180,E1 -7313.192,E2 -7313.192} C_VEL
LIN {X 0,Y 478.074,Z 642.652,A -85,B 0,C 180,E1 -7315.234,E2 -7315.234} C_VEL
LIN {X 0,Y 477.218,Z 636.836,A -85,B 0,C 180,E1 -7316.219,E2 -7316.219} C_VEL
LIN {X 0,Y 474.679,Z 625.483,A -85,B 0,C 180,E1 -7318.28,E2 -7318.28} C_VEL
LIN {X 0,Y 474.601,Z 625.492,A -85,B 0,C 180,E1 -7321.217,E2 -7321.217} C_VEL
LIN {X 0,Y 474.635,Z 625.482,A -85,B 0,C 180,E1 -7324.241,E2 -7324.241} C_VEL
LIN {X 0,Y 474.595,Z 625.494,A -85,B 0,C 180,E1 -7327.383,E2 -7327.383} C_VEL
LIN {X 0,Y 474.644,Z 625.484,A -85,B 0,C 180,E1 -7329.65,E2 -7329.65} C_VEL
LIN {X 0,Y 474.636,Z 625.486,A -85,B 0,C 180,E1 -7332.932,E2 -7332.932} C_VEL
LIN {X 0,Y 474.61,Z 625.489,A -85,B 0,C 180,E1 -7335.895,E2 -7335.895} C_VEL
LIN {X 0,Y 474.642,Z 625.481,A -85,B 0,C 180,E1 -7339.039,E2 -7339.039} C_VEL
LIN {X 0,Y 474.618,Z 625.484,A -85,B 0,C 180,E1 -7341.703,E2 -7341.703} C_VEL
LIN {X 0,Y 474.632,Z 625.483,A -85,B 0,C 180,E1 -7344.726,E2 -7344.726} C_VEL
LIN {X 0,Y 474.638,Z 625.477,A -85,B 0,C 180,E1 -7347.788,E2 -7347.788} C_VEL
LIN {X 0,Y 474.625,Z 625.482,A -85,B 0,C 180,E1 -7350.885,E2 -7350.885} C_VEL
LIN {X 0,Y 474.662,Z 625.483,A -85,B 0,C 180,E1 -7353.629,E2 -7353.629} C_VEL
LIN {X 0,Y 474.637,Z 625.481,A -85,B 0,C 180,E1 -7356.641,E2 -7356.641} C_VEL
LIN {X 0,Y 474.659,Z 625.485,A -85,B 0,C 180,E1 -7360.09,E2 -7360.09} C_VEL
LIN {X 0,Y 474.653,Z 625.48,A -85,B 0,C 180,E1 -7362.775,E2 -7362.775} C_VEL
LIN {X 0,Y 474.65,Z 625.481,A -85,B 0,C 180,E1 -7365.421,E2 -7365.421} C_VEL
LIN {X 0,Y 474.706,Z 625.48,A -85,B 0,C 180,E1 -7368.038,E2 -7368.038} C_VEL
LIN {X 0,Y 474.73,Z 625.468,A -85,B 0,C 180,E1 -7371.487,E2 -7371.487} C_VEL
LIN {X 0,Y 474.775,Z 625.472,A -85,B 0,C 180,E1 -7374.053,E2 -7374.053} C_VEL
LIN {X 0,Y 474.896,Z 625.45,A -85,B 0,C 180,E1 -7377.456,E2 -7377.456} C_VEL
LIN {X 0,Y 474.913,Z 625.451,A -85,B 0,C 180,E1 -7380,E2 -7380} C_VEL
LIN {X 0,Y 474.895,Z 625.457,A -85,B 0,C 180,E1 -7382.545,E2 -7382.545} C_VEL
LIN {X 0,Y 474.772,Z 625.463,A -85,B 0,C 180,E1 -7385.948,E2 -7385.948} C_VEL
LIN {X 0,Y 474.729,Z 625.478,A -85,B 0,C 180,E1 -7388.514,E2 -7388.514} C_VEL
LIN {X 0,Y 474.707,Z 625.474,A -85,B 0,C 180,E1 -7391.963,E2 -7391.963} C_VEL
LIN {X 0,Y 474.703,Z 625.472,A -85,B 0,C 180,E1 -7395.456,E2 -7395.456} C_VEL
LIN {X 0,Y 474.665,Z 625.48,A -85,B 0,C 180,E1 -7399.011,E2 -7399.011} C_VEL
LIN {X 0,Y 474.591,Z 625.489,A -85,B 0,C 180,E1 -7401.729,E2 -7401.729} C_VEL
LIN {X 0,Y 474.652,Z 625.482,A -85,B 0,C 180,E1 -7404.494,E2 -7404.494} C_VEL
LIN {X 0,Y 474.639,Z 625.479,A -85,B 0,C 180,E1 -7407.324,E2 -7407.324} C_VEL
LIN {X 0,Y 474.604,Z 625.48,A -85,B 0,C 180,E1 -7410.231,E2 -7410.231} C_VEL
LIN {X 0,Y 474.627,Z 625.487,A -85,B 0,C 180,E1 -7413.222,E2 -7413.222} C_VEL
LIN {X 0,Y 474.591,Z 625.489,A -85,B 0,C 180,E1 -7416.324,E2 -7416.324} C_VEL
LIN {X 0,Y 474.624,Z 625.483,A -85,B 0,C 180,E1 -7419.548,E2 -7419.548} C_VEL
LIN {X 0,Y 474.588,Z 625.488,A -85,B 0,C 180,E1 -7422.232,E2 -7422.232} C_VEL
LIN {X 0,Y 474.618,Z 625.487,A -85,B 0,C 180,E1 -7425.298,E2 -7425.298} C_VEL
LIN {X 0,Y 474.597,Z 625.49,A -85,B 0,C 180,E1 -7428.212,E2 -7428.212} C_VEL
LIN {X 0,Y 474.612,Z 625.493,A -85,B 0,C 180,E1 -7431.543,E2 -7431.543} C_VEL
LIN {X 0,Y 474.624,Z 625.484,A -85,B 0,C 180,E1 -7434.726,E2 -7434.726} C_VEL
LIN {X 0,Y 474.629,Z 625.483,A -85,B 0,C 180,E1 -7437.787,E2 -7437.787} C_VEL
LIN {X 0,Y 474.621,Z 625.492,A -85,B 0,C 180,E1 -7441.233,E2 -7441.233} C_VEL
LIN {X 0,Y 474.675,Z 625.698,A -85,B 0,C 180,E1 -7441.599,E2 -7441.599} C_VEL
LIN {X 0,Y 476.641,Z 636.012,A -85,B 0,C 180,E1 -7443.746,E2 -7443.746} C_VEL
LIN {X 0,Y 476.546,Z 641.318,A -85,B 0,C 180,E1 -7444.743,E2 -7444.743} C_VEL
LIN {X 0,Y 480.138,Z 657.755,A -85,B 0,C 180,E1 -7445.166,E2 -7445.166} C_VEL
LIN {X 0,Y 480.147,Z 672.046,A -85,B 0,C 180,E1 -7445.391,E2 -7445.391} C_VEL
LIN {X 0,Y 479.441,Z 677.893,A -85,B 0,C 180,E1 -7445.451,E2 -7445.451} C_VEL
LIN {X 0,Y 473.846,Z 696.923,A -85,B 0,C 180,E1 -7445.5,E2 -7445.5} C_VEL
LIN {X 0,Y 473.154,Z 702.769,A -85,B 0,C 180,E1 -7445.562,E2 -7445.562} C_VEL
LIN {X 0,Y 472.48,Z 777.083,A -85,B 0,C 180,E1 -7446.727,E2 -7446.727} C_VEL
LIN {X 0,Y 472.121,Z 791.431,A -85,B 0,C 180,E1 -7447.114,E2 -7447.114} C_VEL
LIN {X 0,Y 471.541,Z 805.033,A -85,B 0,C 180,E1 -7447.652,E2 -7447.652} C_VEL
LIN {X 0,Y 470.997,Z 817.75,A -85,B 0,C 180,E1 -7448.327,E2 -7448.327} C_VEL
LIN {X 0,Y 470.328,Z 830.79,A -85,B 0,C 180,E1 -7449.213,E2 -7449.213} C_VEL
LIN {X 0,Y 469.688,Z 842.494,A -85,B 0,C 180,E1 -7450.204,E2 -7450.204} C_VEL
LIN {X 0,Y 469.111,Z 852.34,A -85,B 0,C 180,E1 -7451.21,E2 -7451.21} C_VEL
LIN {X 0,Y 468.444,Z 863.121,A -85,B 0,C 180,E1 -7452.539,E2 -7452.539} C_VEL
LIN {X 0,Y 467.901,Z 872.845,A -85,B 0,C 180,E1 -7454.009,E2 -7454.009} C_VEL
LIN {X 0,Y 467.441,Z 880.424,A -85,B 0,C 180,E1 -7455.414,E2 -7455.414} C_VEL
LIN {X 0,Y 467.123,Z 887.173,A -85,B 0,C 180,E1 -7456.957,E2 -7456.957} C_VEL
LIN {X 0,Y 466.846,Z 893.119,A -85,B 0,C 180,E1 -7458.714,E2 -7458.714} C_VEL
LIN {X 0,Y 466.692,Z 897.457,A -85,B 0,C 180,E1 -7460.465,E2 -7460.465} C_VEL
LIN {X 0,Y 466.654,Z 900.329,A -85,B 0,C 180,E1 -7462.21,E2 -7462.21} C_VEL
LIN {X 0,Y 466.645,Z 901.829,A -85,B 0,C 180,E1 -7463.948,E2 -7463.948} C_VEL
LIN {X 0,Y 466.589,Z 902.007,A -85,B 0,C 180,E1 -7465.681,E2 -7465.681} C_VEL
LIN {X 0,Y 466.691,Z 901.599,A -85,B 0,C 180,E1 -7466.547,E2 -7466.547} C_VEL
LIN {X 0,Y 466.689,Z 899.807,A -85,B 0,C 180,E1 -7468.274,E2 -7468.274} C_VEL
LIN {X 0,Y 466.632,Z 896.672,A -85,B 0,C 180,E1 -7470,E2 -7470} C_VEL
LIN {X 0,Y 466.761,Z 892.066,A -85,B 0,C 180,E1 -7471.726,E2 -7471.726} C_VEL
LIN {X 0,Y 467.157,Z 885.849,A -85,B 0,C 180,E1 -7473.45,E2 -7473.45} C_VEL
LIN {X 0,Y 467.562,Z 878.948,A -85,B 0,C 180,E1 -7474.958,E2 -7474.958} C_VEL
LIN {X 0,Y 467.951,Z 871.757,A -85,B 0,C 180,E1 -7476.251,E2 -7476.251} C_VEL
LIN {X 0,Y 468.441,Z 863.127,A -85,B 0,C 180,E1 -7477.543,E2 -7477.543} C_VEL
LIN {X 0,Y 469.089,Z 852.685,A -85,B 0,C 180,E1 -7478.834,E2 -7478.834} C_VEL
LIN {X 0,Y 469.797,Z 841.002,A -85,B 0,C 180,E1 -7480.015,E2 -7480.015} C_VEL
LIN {X 0,Y 470.405,Z 829.277,A -85,B 0,C 180,E1 -7480.981,E2 -7480.981} C_VEL
LIN {X 0,Y 471.147,Z 816.305,A -85,B 0,C 180,E1 -7481.836,E2 -7481.836} C_VEL
LIN {X 0,Y 471.699,Z 802.627,A -85,B 0,C 180,E1 -7482.531,E2 -7482.531} C_VEL
LIN {X 0,Y 472.093,Z 789.046,A -85,B 0,C 180,E1 -7483.04,E2 -7483.04} C_VEL
LIN {X 0,Y 472.338,Z 775.163,A -85,B 0,C 180,E1 -7483.389,E2 -7483.389} C_VEL
LIN {X 0,Y 473.461,Z 658.815,A -85,B 0,C 180,E1 -7485.186,E2 -7485.186} C_VEL
LIN {X 0,Y 469.619,Z 641.258,A -85,B 0,C 180,E1 -7485.655,E2 -7485.655} C_VEL
LIN {X 0,Y 469.526,Z 636.054,A -85,B 0,C 180,E1 -7486.669,E2 -7486.669} C_VEL
LIN {X 0,Y 467.613,Z 626.367,A -85,B 0,C 180,E1 -7488.723,E2 -7488.723} C_VEL
LIN {X 0,Y 467.585,Z 626.367,A -85,B 0,C 180,E1 -7491.268,E2 -7491.268} C_VEL
LIN {X 0,Y 467.556,Z 626.368,A -85,B 0,C 180,E1 -7493.944,E2 -7493.944} C_VEL
LIN {X 0,Y 467.528,Z 626.375,A -85,B 0,C 180,E1 -7496.806,E2 -7496.806} C_VEL
LIN {X 0,Y 467.535,Z 626.369,A -85,B 0,C 180,E1 -7499.74,E2 -7499.74} C_VEL
LIN {X 0,Y 467.551,Z 626.373,A -85,B 0,C 180,E1 -7502.761,E2 -7502.761} C_VEL
LIN {X 0,Y 467.546,Z 626.366,A -85,B 0,C 180,E1 -7505.891,E2 -7505.891} C_VEL
